LIN {X 0.040,Y -457.437,Z 279.553,A 0.000,B 0.000,C 90.000,E1 279.500} C_DIS
LIN {X 0.163,Y -463.352,Z 279.547,A 0.000,B 0.000,C 90.000,E1 278.454} C_DIS
LIN {X -0.027,Y -471.556,Z 279.539,A 0.000,B 0.000,C 90.000,E1 276.947} C_DIS
LIN {X 0.196,Y -476.547,Z 279.533,A 0.000,B 0.000,C 90.000,E1 275.910} C_DIS
LIN {X -0.146,Y -478.748,Z 279.530,A 0.000,B 0.000,C 90.000,E1 275.448} C_DIS
LIN {X -0.043,Y -480.665,Z 279.527,A 0.000,B 0.000,C 90.000,E1 274.935} C_DIS
LIN {X 0.113,Y -482.200,Z 279.525,A 0.000,B 0.000,C 90.000,E1 274.416} C_DIS
LIN {X -0.205,Y -483.358,Z 279.522,A 0.000,B 0.000,C 90.000,E1 273.955} C_DIS
LIN {X -0.065,Y -484.126,Z 279.519,A 0.000,B 0.000,C 90.000,E1 273.440} C_DIS
LIN {X 0.111,Y -484.567,Z 279.516,A 0.000,B 0.000,C 90.000,E1 272.922} C_DIS
LIN {X -0.218,Y -484.699,Z 279.514,A 0.000,B 0.000,C 90.000,E1 272.465} C_DIS
LIN {X 0.119,Y -484.413,Z 279.508,A 0.000,B 0.000,C 90.000,E1 271.432} C_DIS
LIN {X -0.203,Y -484.109,Z 279.505,A 0.000,B 0.000,C 90.000,E1 270.974} C_DIS
LIN {X -0.042,Y -483.584,Z 279.503,A 0.000,B 0.000,C 90.000,E1 270.458} C_DIS
LIN {X 0.119,Y -482.708,Z 279.500,A 0.000,B 0.000,C 90.000,E1 269.943} C_DIS
LIN {X -0.206,Y -481.433,Z 279.497,A 0.000,B 0.000,C 90.000,E1 269.484} C_DIS
LIN {X -0.056,Y -479.640,Z 279.494,A 0.000,B 0.000,C 90.000,E1 268.969} C_DIS
LIN {X 0.085,Y -477.139,Z 279.491,A 0.000,B 0.000,C 90.000,E1 268.453} C_DIS
LIN {X 0.223,Y -473.997,Z 279.489,A 0.000,B 0.000,C 90.000,E1 267.936} C_DIS
LIN {X -0.142,Y -469.925,Z 279.486,A 0.000,B 0.000,C 90.000,E1 267.478} C_DIS
LIN {X 0.134,Y -467.510,Z 279.484,A 0.000,B 0.000,C 90.000,E1 267.192} C_DIS
LIN {X -0.099,Y -461.974,Z 279.482,A 0.000,B 0.000,C 90.000,E1 266.731} C_DIS
LIN {X -0.164,Y -458.751,Z 279.480,A 0.000,B 0.000,C 90.000,E1 266.502} C_DIS
LIN {X 0.047,Y -455.605,Z 279.479,A 0.000,B 0.000,C 90.000,E1 266.274} C_DIS
LIN {X -0.198,Y -451.886,Z 279.478,A 0.000,B 0.000,C 90.000,E1 266.102} C_DIS
LIN {X -0.075,Y -448.465,Z 279.477,A 0.000,B 0.000,C 90.000,E1 265.927} C_DIS
LIN {X 0.016,Y -444.357,Z 279.476,A 0.000,B 0.000,C 90.000,E1 265.755} C_DIS
LIN {X -0.022,Y -440.666,Z 279.476,A 0.000,B 0.000,C 90.000,E1 265.641} C_DIS
LIN {X -0.059,Y -435.858,Z 279.475,A 0.000,B 0.000,C 90.000,E1 265.527} C_DIS
LIN {X 0.058,Y -425.990,Z 279.474,A 0.000,B 0.000,C 90.000,E1 265.355} C_DIS
LIN {X 0.041,Y -418.591,Z 279.474,A 0.000,B 0.000,C 90.000,E1 265.298} C_DIS
LIN {X -0.001,Y -180.904,Z 279.474,A 0.000,B 0.000,C 90.000,E1 265.298} C_DIS
LIN {X 0.035,Y -180.229,Z 279.464,A 0.000,B 0.000,C 90.000,E1 263.571} C_DIS
LIN {X -0.012,Y -179.042,Z 279.446,A 0.000,B 0.000,C 90.000,E1 260.208} C_DIS
LIN {X 0.051,Y -178.713,Z 279.441,A 0.000,B 0.000,C 90.000,E1 259.342} C_DIS
LIN {X -0.056,Y -175.761,Z 279.413,A 0.000,B 0.000,C 90.000,E1 254.283} C_DIS
LIN {X -0.006,Y -171.945,Z 279.384,A 0.000,B 0.000,C 90.000,E1 249.135} C_DIS
LIN {X -0.030,Y -171.330,Z 279.379,A 0.000,B 0.000,C 90.000,E1 248.284} C_DIS
LIN {X 0.022,Y -167.585,Z 279.355,A 0.000,B 0.000,C 90.000,E1 243.948} C_DIS
LIN {X -0.039,Y -166.222,Z 279.346,A 0.000,B 0.000,C 90.000,E1 242.231} C_DIS
LIN {X -0.050,Y -162.984,Z 279.326,A 0.000,B 0.000,C 90.000,E1 238.742} C_DIS
LIN {X -0.003,Y -160.899,Z 279.312,A 0.000,B 0.000,C 90.000,E1 236.087} C_DIS
LIN {X -0.025,Y -157.667,Z 279.292,A 0.000,B 0.000,C 90.000,E1 232.557} C_DIS
LIN {X -0.086,Y -155.705,Z 279.277,A 0.000,B 0.000,C 90.000,E1 229.908} C_DIS
LIN {X -0.032,Y -151.967,Z 279.252,A 0.000,B 0.000,C 90.000,E1 225.405} C_DIS
LIN {X -0.015,Y -150.210,Z 279.237,A 0.000,B 0.000,C 90.000,E1 222.690} C_DIS
LIN {X -0.090,Y -146.976,Z 279.212,A 0.000,B 0.000,C 90.000,E1 218.177} C_DIS
LIN {X 0.019,Y -145.562,Z 279.197,A 0.000,B 0.000,C 90.000,E1 215.391} C_DIS
LIN {X 0.018,Y -142.954,Z 279.171,A 0.000,B 0.000,C 90.000,E1 210.797} C_DIS
LIN {X -0.051,Y -141.580,Z 279.151,A 0.000,B 0.000,C 90.000,E1 207.129} C_DIS
LIN {X -0.003,Y -139.415,Z 279.115,A 0.000,B 0.000,C 90.000,E1 200.610} C_DIS
LIN {X 0.048,Y -139.140,Z 279.104,A 0.000,B 0.000,C 90.000,E1 198.725} C_DIS
LIN {X -0.061,Y -138.348,Z 279.057,A 0.000,B 0.000,C 90.000,E1 190.366} C_DIS
LIN {X 0.063,Y -139.492,Z 279.006,A 0.000,B 0.000,C 90.000,E1 180.974} C_DIS
LIN {X 0.004,Y -141.103,Z 278.975,A 0.000,B 0.000,C 90.000,E1 175.412} C_DIS
LIN {X -0.043,Y -142.482,Z 278.959,A 0.000,B 0.000,C 90.000,E1 172.648} C_DIS
LIN {X 0.047,Y -144.731,Z 278.933,A 0.000,B 0.000,C 90.000,E1 167.993} C_DIS
LIN {X -0.003,Y -147.335,Z 278.913,A 0.000,B 0.000,C 90.000,E1 164.338} C_DIS
LIN {X 0.062,Y -150.658,Z 278.888,A 0.000,B 0.000,C 90.000,E1 159.752} C_DIS
LIN {X -0.056,Y -154.136,Z 278.868,A 0.000,B 0.000,C 90.000,E1 156.177} C_DIS
LIN {X 0.006,Y -157.565,Z 278.848,A 0.000,B 0.000,C 90.000,E1 152.564} C_DIS
LIN {X 0.030,Y -161.808,Z 278.828,A 0.000,B 0.000,C 90.000,E1 148.997} C_DIS
LIN {X 0.050,Y -166.000,Z 278.808,A 0.000,B 0.000,C 90.000,E1 145.468} C_DIS
LIN {X 0.042,Y -170.999,Z 278.789,A 0.000,B 0.000,C 90.000,E1 141.984} C_DIS
LIN {X -0.042,Y -175.868,Z 278.770,A 0.000,B 0.000,C 90.000,E1 138.566} C_DIS
LIN {X -0.049,Y -181.473,Z 278.751,A 0.000,B 0.000,C 90.000,E1 135.162} C_DIS
LIN {X 0.088,Y -186.986,Z 278.732,A 0.000,B 0.000,C 90.000,E1 131.757} C_DIS
LIN {X 0.090,Y -190.102,Z 278.723,A 0.000,B 0.000,C 90.000,E1 130.092} C_DIS
LIN {X 0.110,Y -195.874,Z 278.705,A 0.000,B 0.000,C 90.000,E1 126.790} C_DIS
LIN {X -0.098,Y -200.705,Z 278.691,A 0.000,B 0.000,C 90.000,E1 124.405} C_DIS
LIN {X 0.009,Y -203.178,Z 278.683,A 0.000,B 0.000,C 90.000,E1 122.959} C_DIS
LIN {X -0.023,Y -305.671,Z 278.683,A 0.000,B 0.000,C 90.000,E1 122.959} C_DIS
LIN {X 0.050,Y -311.024,Z 278.682,A 0.000,B 0.000,C 90.000,E1 122.752} C_DIS
LIN {X 0.065,Y -314.178,Z 278.681,A 0.000,B 0.000,C 90.000,E1 122.498} C_DIS
LIN {X -0.074,Y -317.883,Z 278.678,A 0.000,B 0.000,C 90.000,E1 122.054} C_DIS
LIN {X -0.012,Y -319.669,Z 278.676,A 0.000,B 0.000,C 90.000,E1 121.720} C_DIS
LIN {X -0.034,Y -322.247,Z 278.673,A 0.000,B 0.000,C 90.000,E1 121.082} C_DIS
LIN {X -0.019,Y -333.580,Z 278.657,A 0.000,B 0.000,C 90.000,E1 118.231} C_DIS
LIN {X -0.161,Y -346.345,Z 278.641,A 0.000,B 0.000,C 90.000,E1 115.463} C_DIS
LIN {X -0.119,Y -358.992,Z 278.628,A 0.000,B 0.000,C 90.000,E1 113.025} C_DIS
LIN {X 0.117,Y -372.959,Z 278.615,A 0.000,B 0.000,C 90.000,E1 110.610} C_DIS
LIN {X -0.037,Y -388.346,Z 278.602,A 0.000,B 0.000,C 90.000,E1 108.308} C_DIS
LIN {X 0.072,Y -405.270,Z 278.589,A 0.000,B 0.000,C 90.000,E1 106.024} C_DIS
LIN {X -0.019,Y -423.855,Z 278.577,A 0.000,B 0.000,C 90.000,E1 103.828} C_DIS
LIN {X 0.042,Y -443.818,Z 278.565,A 0.000,B 0.000,C 90.000,E1 101.715} C_DIS
LIN {X -0.025,Y -464.375,Z 278.554,A 0.000,B 0.000,C 90.000,E1 99.792} C_DIS
LIN {X -0.069,Y -488.109,Z 278.543,A 0.000,B 0.000,C 90.000,E1 97.814} C_DIS
LIN {X 0.073,Y -501.323,Z 278.538,A 0.000,B 0.000,C 90.000,E1 96.777} C_DIS
LIN {X -0.176,Y -503.227,Z 278.537,A 0.000,B 0.000,C 90.000,E1 96.606} C_DIS
LIN {X 0.250,Y -504.994,Z 278.535,A 0.000,B 0.000,C 90.000,E1 96.315} C_DIS
LIN {X 0.120,Y -506.320,Z 278.534,A 0.000,B 0.000,C 90.000,E1 96.087} C_DIS
LIN {X -0.066,Y -507.964,Z 278.531,A 0.000,B 0.000,C 90.000,E1 95.625} C_DIS
LIN {X -0.247,Y -508.512,Z 278.529,A 0.000,B 0.000,C 90.000,E1 95.163} C_DIS
LIN {X 0.086,Y -508.054,Z 278.526,A 0.000,B 0.000,C 90.000,E1 94.645} C_DIS
LIN {X -0.125,Y -506.510,Z 278.523,A 0.000,B 0.000,C 90.000,E1 94.188} C_DIS
LIN {X -0.194,Y -505.243,Z 278.522,A 0.000,B 0.000,C 90.000,E1 93.955} C_DIS
LIN {X 0.093,Y -501.741,Z 278.519,A 0.000,B 0.000,C 90.000,E1 93.440} C_DIS
LIN {X 0.140,Y -493.907,Z 278.514,A 0.000,B 0.000,C 90.000,E1 92.465} C_DIS
LIN {X -0.053,Y -483.305,Z 278.507,A 0.000,B 0.000,C 90.000,E1 91.260} C_DIS
LIN {X -0.212,Y -464.590,Z 278.494,A 0.000,B 0.000,C 90.000,E1 89.026} C_DIS
LIN {X 0.122,Y -451.376,Z 278.484,A 0.000,B 0.000,C 90.000,E1 87.192} C_DIS
LIN {X 0.186,Y -430.844,Z 278.467,A 0.000,B 0.000,C 90.000,E1 84.033} C_DIS
LIN {X -0.180,Y -416.871,Z 278.454,A 0.000,B 0.000,C 90.000,E1 81.659} C_DIS
LIN {X 0.002,Y -404.089,Z 278.440,A 0.000,B 0.000,C 90.000,E1 79.162} C_DIS
LIN {X -0.157,Y -394.044,Z 278.429,A 0.000,B 0.000,C 90.000,E1 77.229} C_DIS
LIN {X -0.017,Y -382.646,Z 278.416,A 0.000,B 0.000,C 90.000,E1 74.936} C_DIS
LIN {X 0.035,Y -374.165,Z 278.407,A 0.000,B 0.000,C 90.000,E1 73.196} C_DIS
LIN {X -0.012,Y -362.792,Z 278.394,A 0.000,B 0.000,C 90.000,E1 70.859} C_DIS
LIN {X 0.068,Y -350.331,Z 278.379,A 0.000,B 0.000,C 90.000,E1 68.156} C_DIS
LIN {X 0.070,Y -336.135,Z 278.360,A 0.000,B 0.000,C 90.000,E1 64.793} C_DIS
LIN {X -0.024,Y -322.120,Z 278.339,A 0.000,B 0.000,C 90.000,E1 61.051} C_DIS
LIN {X 0.127,Y -314.316,Z 278.327,A 0.000,B 0.000,C 90.000,E1 58.791} C_DIS
LIN {X 0.061,Y -305.742,Z 278.312,A 0.000,B 0.000,C 90.000,E1 56.215} C_DIS
LIN {X -0.112,Y -297.454,Z 278.298,A 0.000,B 0.000,C 90.000,E1 53.623} C_DIS
LIN {X 0.045,Y -289.244,Z 278.283,A 0.000,B 0.000,C 90.000,E1 50.928} C_DIS
LIN {X -0.099,Y -283.046,Z 278.272,A 0.000,B 0.000,C 90.000,E1 48.933} C_DIS
LIN {X 0.000,Y -272.943,Z 278.253,A 0.000,B 0.000,C 90.000,E1 45.486} C_DIS
LIN {X 0.038,Y -265.369,Z 278.237,A 0.000,B 0.000,C 90.000,E1 42.690} C_DIS
LIN {X -0.178,Y -259.814,Z 278.225,A 0.000,B 0.000,C 90.000,E1 40.620} C_DIS
LIN {X -0.101,Y -254.173,Z 278.214,A 0.000,B 0.000,C 90.000,E1 38.463} C_DIS
LIN {X -0.091,Y -248.423,Z 278.202,A 0.000,B 0.000,C 90.000,E1 36.297} C_DIS
LIN {X 0.064,Y -242.506,Z 278.189,A 0.000,B 0.000,C 90.000,E1 34.072} C_DIS
LIN {X -0.015,Y -232.916,Z 278.169,A 0.000,B 0.000,C 90.000,E1 30.384} C_DIS
LIN {X -0.085,Y -225.892,Z 278.152,A 0.000,B 0.000,C 90.000,E1 27.385} C_DIS
LIN {X -0.125,Y -219.659,Z 278.135,A 0.000,B 0.000,C 90.000,E1 24.335} C_DIS
LIN {X -0.029,Y -212.898,Z 278.113,A 0.000,B 0.000,C 90.000,E1 20.429} C_DIS
LIN {X -0.041,Y -207.094,Z 278.092,A 0.000,B 0.000,C 90.000,E1 16.496} C_DIS
LIN {X 0.077,Y -202.346,Z 278.069,A 0.000,B 0.000,C 90.000,E1 12.479} C_DIS
LIN {X 0.079,Y -198.629,Z 278.047,A 0.000,B 0.000,C 90.000,E1 8.454} C_DIS
LIN {X -0.050,Y -195.024,Z 278.016,A 0.000,B 0.000,C 90.000,E1 2.808} C_DIS
LIN {X 0.076,Y -195.799,Z 277.920,A 0.000,B 0.000,C 90.000,E1 345.589} C_DIS
LIN {X -0.008,Y -199.281,Z 277.893,A 0.000,B 0.000,C 90.000,E1 340.732} C_DIS
LIN {X 0.093,Y -203.362,Z 277.871,A 0.000,B 0.000,C 90.000,E1 336.666} C_DIS
LIN {X 0.003,Y -208.478,Z 277.848,A 0.000,B 0.000,C 90.000,E1 332.692} C_DIS
LIN {X -0.007,Y -214.658,Z 277.826,A 0.000,B 0.000,C 90.000,E1 328.742} C_DIS
LIN {X 0.080,Y -220.531,Z 277.809,A 0.000,B 0.000,C 90.000,E1 325.595} C_DIS
LIN {X -0.106,Y -227.213,Z 277.792,A 0.000,B 0.000,C 90.000,E1 322.557} C_DIS
LIN {X 0.076,Y -235.809,Z 277.773,A 0.000,B 0.000,C 90.000,E1 319.094} C_DIS
LIN {X 0.137,Y -245.410,Z 277.754,A 0.000,B 0.000,C 90.000,E1 315.729} C_DIS
LIN {X 0.135,Y -256.023,Z 277.736,A 0.000,B 0.000,C 90.000,E1 312.447} C_DIS
LIN {X -0.070,Y -267.676,Z 277.718,A 0.000,B 0.000,C 90.000,E1 309.277} C_DIS
LIN {X 0.151,Y -280.621,Z 277.701,A 0.000,B 0.000,C 90.000,E1 306.091} C_DIS
LIN {X 0.116,Y -293.578,Z 277.686,A 0.000,B 0.000,C 90.000,E1 303.372} C_DIS
LIN {X -0.041,Y -309.906,Z 277.669,A 0.000,B 0.000,C 90.000,E1 300.413} C_DIS
LIN {X 0.048,Y -329.857,Z 277.651,A 0.000,B 0.000,C 90.000,E1 297.180} C_DIS
LIN {X -0.144,Y -342.555,Z 277.641,A 0.000,B 0.000,C 90.000,E1 295.335} C_DIS
LIN {X 0.074,Y -355.273,Z 277.630,A 0.000,B 0.000,C 90.000,E1 293.462} C_DIS
LIN {X 0.079,Y -368.073,Z 277.620,A 0.000,B 0.000,C 90.000,E1 291.663} C_DIS
LIN {X 0.078,Y -385.539,Z 277.607,A 0.000,B 0.000,C 90.000,E1 289.322} C_DIS
LIN {X 0.060,Y -401.077,Z 277.596,A 0.000,B 0.000,C 90.000,E1 287.330} C_DIS
LIN {X 0.024,Y -414.297,Z 277.587,A 0.000,B 0.000,C 90.000,E1 285.662} C_DIS
LIN {X -0.034,Y -425.272,Z 277.579,A 0.000,B 0.000,C 90.000,E1 284.300} C_DIS
LIN {X 0.039,Y -431.512,Z 277.575,A 0.000,B 0.000,C 90.000,E1 283.480} C_DIS
LIN {X 0.038,Y -439.105,Z 277.569,A 0.000,B 0.000,C 90.000,E1 282.411} C_DIS
LIN {X 0.163,Y -447.753,Z 277.562,A 0.000,B 0.000,C 90.000,E1 281.074} C_DIS
LIN {X -0.014,Y -455.691,Z 277.554,A 0.000,B 0.000,C 90.000,E1 279.792} C_DIS
LIN {X 0.089,Y -461.705,Z 277.549,A 0.000,B 0.000,C 90.000,E1 278.746} C_DIS
LIN {X 0.035,Y -468.676,Z 277.542,A 0.000,B 0.000,C 90.000,E1 277.473} C_DIS
LIN {X -0.186,Y -473.921,Z 277.536,A 0.000,B 0.000,C 90.000,E1 276.486} C_DIS
LIN {X 0.017,Y -478.571,Z 277.530,A 0.000,B 0.000,C 90.000,E1 275.454} C_DIS
LIN {X 0.166,Y -480.481,Z 277.528,A 0.000,B 0.000,C 90.000,E1 274.935} C_DIS
LIN {X -0.160,Y -482.031,Z 277.525,A 0.000,B 0.000,C 90.000,E1 274.473} C_DIS
LIN {X 0.002,Y -483.221,Z 277.522,A 0.000,B 0.000,C 90.000,E1 273.955} C_DIS
LIN {X 0.141,Y -483.997,Z 277.519,A 0.000,B 0.000,C 90.000,E1 273.440} C_DIS
LIN {X -0.167,Y -484.471,Z 277.516,A 0.000,B 0.000,C 90.000,E1 272.980} C_DIS
LIN {X -0.013,Y -484.651,Z 277.514,A 0.000,B 0.000,C 90.000,E1 272.465} C_DIS
LIN {X 0.148,Y -484.631,Z 277.511,A 0.000,B 0.000,C 90.000,E1 271.949} C_DIS
LIN {X 0.001,Y -484.162,Z 277.505,A 0.000,B 0.000,C 90.000,E1 270.974} C_DIS
LIN {X 0.163,Y -483.651,Z 277.503,A 0.000,B 0.000,C 90.000,E1 270.458} C_DIS
LIN {X -0.160,Y -482.807,Z 277.500,A 0.000,B 0.000,C 90.000,E1 270.000} C_DIS
LIN {X -0.002,Y -481.535,Z 277.497,A 0.000,B 0.000,C 90.000,E1 269.484} C_DIS
LIN {X 0.148,Y -479.754,Z 277.494,A 0.000,B 0.000,C 90.000,E1 268.969} C_DIS
LIN {X -0.188,Y -477.339,Z 277.492,A 0.000,B 0.000,C 90.000,E1 268.511} C_DIS
LIN {X -0.048,Y -474.199,Z 277.489,A 0.000,B 0.000,C 90.000,E1 267.993} C_DIS
LIN {X 0.061,Y -470.202,Z 277.486,A 0.000,B 0.000,C 90.000,E1 267.478} C_DIS
LIN {X 0.143,Y -465.186,Z 277.483,A 0.000,B 0.000,C 90.000,E1 266.963} C_DIS
LIN {X 0.067,Y -462.356,Z 277.482,A 0.000,B 0.000,C 90.000,E1 266.731} C_DIS
LIN {X -0.032,Y -459.122,Z 277.481,A 0.000,B 0.000,C 90.000,E1 266.502} C_DIS
LIN {X 0.161,Y -455.979,Z 277.479,A 0.000,B 0.000,C 90.000,E1 266.274} C_DIS
LIN {X -0.003,Y -449.020,Z 277.477,A 0.000,B 0.000,C 90.000,E1 265.927} C_DIS
LIN {X 0.061,Y -444.993,Z 277.476,A 0.000,B 0.000,C 90.000,E1 265.755} C_DIS
LIN {X -0.081,Y -436.493,Z 277.475,A 0.000,B 0.000,C 90.000,E1 265.527} C_DIS
LIN {X 0.150,Y -432.276,Z 277.475,A 0.000,B 0.000,C 90.000,E1 265.412} C_DIS
LIN {X -0.049,Y -426.466,Z 277.474,A 0.000,B 0.000,C 90.000,E1 265.355} C_DIS
LIN {X -0.056,Y -419.057,Z 277.474,A 0.000,B 0.000,C 90.000,E1 265.298} C_DIS
LIN {X -0.104,Y -416.418,Z 277.474,A 0.000,B 0.000,C 90.000,E1 265.298} C_DIS
LIN {X -0.066,Y -180.902,Z 277.474,A 0.000,B 0.000,C 90.000,E1 265.298} C_DIS
LIN {X -0.018,Y -180.222,Z 277.464,A 0.000,B 0.000,C 90.000,E1 263.571} C_DIS
LIN {X -0.065,Y -179.037,Z 277.445,A 0.000,B 0.000,C 90.000,E1 260.208} C_DIS
LIN {X -0.002,Y -178.701,Z 277.441,A 0.000,B 0.000,C 90.000,E1 259.342} C_DIS
LIN {X -0.061,Y -175.751,Z 277.412,A 0.000,B 0.000,C 90.000,E1 254.267} C_DIS
LIN {X -0.058,Y -171.934,Z 277.384,A 0.000,B 0.000,C 90.000,E1 249.135} C_DIS
LIN {X -0.082,Y -171.314,Z 277.379,A 0.000,B 0.000,C 90.000,E1 248.284} C_DIS
LIN {X -0.028,Y -167.573,Z 277.355,A 0.000,B 0.000,C 90.000,E1 243.948} C_DIS
LIN {X -0.089,Y -166.203,Z 277.346,A 0.000,B 0.000,C 90.000,E1 242.231} C_DIS
LIN {X -0.100,Y -162.969,Z 277.326,A 0.000,B 0.000,C 90.000,E1 238.742} C_DIS
LIN {X -0.052,Y -160.881,Z 277.311,A 0.000,B 0.000,C 90.000,E1 236.087} C_DIS
LIN {X -0.073,Y -157.652,Z 277.292,A 0.000,B 0.000,C 90.000,E1 232.557} C_DIS
LIN {X 0.085,Y -155.689,Z 277.277,A 0.000,B 0.000,C 90.000,E1 229.828} C_DIS
LIN {X -0.079,Y -151.955,Z 277.252,A 0.000,B 0.000,C 90.000,E1 225.405} C_DIS
LIN {X -0.062,Y -150.195,Z 277.237,A 0.000,B 0.000,C 90.000,E1 222.690} C_DIS
LIN {X 0.069,Y -146.965,Z 277.212,A 0.000,B 0.000,C 90.000,E1 218.096} C_DIS
LIN {X -0.028,Y -145.552,Z 277.197,A 0.000,B 0.000,C 90.000,E1 215.391} C_DIS
LIN {X -0.028,Y -142.945,Z 277.171,A 0.000,B 0.000,C 90.000,E1 210.797} C_DIS
LIN {X 0.029,Y -141.571,Z 277.150,A 0.000,B 0.000,C 90.000,E1 207.078} C_DIS
LIN {X -0.049,Y -139.412,Z 277.114,A 0.000,B 0.000,C 90.000,E1 200.610} C_DIS
LIN {X 0.003,Y -139.135,Z 277.104,A 0.000,B 0.000,C 90.000,E1 198.725} C_DIS
LIN {X 0.030,Y -138.349,Z 277.057,A 0.000,B 0.000,C 90.000,E1 190.310} C_DIS
LIN {X 0.018,Y -139.494,Z 277.005,A 0.000,B 0.000,C 90.000,E1 180.974} C_DIS
LIN {X -0.042,Y -141.110,Z 276.974,A 0.000,B 0.000,C 90.000,E1 175.412} C_DIS
LIN {X 0.052,Y -142.490,Z 276.959,A 0.000,B 0.000,C 90.000,E1 172.591} C_DIS
LIN {X 0.000,Y -144.742,Z 276.933,A 0.000,B 0.000,C 90.000,E1 167.993} C_DIS
LIN {X -0.050,Y -147.349,Z 276.913,A 0.000,B 0.000,C 90.000,E1 164.338} C_DIS
LIN {X 0.014,Y -150.674,Z 276.888,A 0.000,B 0.000,C 90.000,E1 159.752} C_DIS
LIN {X 0.035,Y -154.154,Z 276.867,A 0.000,B 0.000,C 90.000,E1 156.125} C_DIS
LIN {X 0.029,Y -157.584,Z 276.848,A 0.000,B 0.000,C 90.000,E1 152.538} C_DIS
LIN {X -0.020,Y -161.832,Z 276.828,A 0.000,B 0.000,C 90.000,E1 148.997} C_DIS
LIN {X -0.001,Y -166.023,Z 276.808,A 0.000,B 0.000,C 90.000,E1 145.468} C_DIS
LIN {X -0.009,Y -171.024,Z 276.789,A 0.000,B 0.000,C 90.000,E1 141.984} C_DIS
LIN {X 0.022,Y -175.894,Z 276.770,A 0.000,B 0.000,C 90.000,E1 138.528} C_DIS
LIN {X 0.026,Y -181.499,Z 276.751,A 0.000,B 0.000,C 90.000,E1 135.121} C_DIS
LIN {X 0.033,Y -187.016,Z 276.732,A 0.000,B 0.000,C 90.000,E1 131.757} C_DIS
LIN {X 0.035,Y -190.134,Z 276.723,A 0.000,B 0.000,C 90.000,E1 130.092} C_DIS
LIN {X 0.053,Y -195.905,Z 276.704,A 0.000,B 0.000,C 90.000,E1 126.790} C_DIS
LIN {X 0.010,Y -200.736,Z 276.691,A 0.000,B 0.000,C 90.000,E1 124.358} C_DIS
LIN {X 0.023,Y -203.258,Z 276.683,A 0.000,B 0.000,C 90.000,E1 122.911} C_DIS
LIN {X 0.166,Y -305.477,Z 276.683,A 0.000,B 0.000,C 90.000,E1 122.880} C_DIS
LIN {X 0.096,Y -306.527,Z 276.683,A 0.000,B 0.000,C 90.000,E1 122.880} C_DIS
LIN {X -0.037,Y -310.653,Z 276.682,A 0.000,B 0.000,C 90.000,E1 122.752} C_DIS
LIN {X -0.175,Y -313.783,Z 276.681,A 0.000,B 0.000,C 90.000,E1 122.546} C_DIS
LIN {X -0.051,Y -317.498,Z 276.678,A 0.000,B 0.000,C 90.000,E1 122.084} C_DIS
LIN {X 0.045,Y -319.375,Z 276.676,A 0.000,B 0.000,C 90.000,E1 121.750} C_DIS
LIN {X -0.131,Y -320.846,Z 276.675,A 0.000,B 0.000,C 90.000,E1 121.465} C_DIS
LIN {X -0.050,Y -333.366,Z 276.657,A 0.000,B 0.000,C 90.000,E1 118.281} C_DIS
LIN {X 0.106,Y -346.106,Z 276.642,A 0.000,B 0.000,C 90.000,E1 115.463} C_DIS
LIN {X -0.179,Y -358.730,Z 276.628,A 0.000,B 0.000,C 90.000,E1 113.078} C_DIS
LIN {X 0.042,Y -372.672,Z 276.615,A 0.000,B 0.000,C 90.000,E1 110.663} C_DIS
LIN {X -0.128,Y -388.033,Z 276.602,A 0.000,B 0.000,C 90.000,E1 108.362} C_DIS
LIN {X -0.035,Y -404.928,Z 276.589,A 0.000,B 0.000,C 90.000,E1 106.079} C_DIS
LIN {X -0.145,Y -423.483,Z 276.577,A 0.000,B 0.000,C 90.000,E1 103.883} C_DIS
LIN {X -0.117,Y -443.431,Z 276.565,A 0.000,B 0.000,C 90.000,E1 101.771} C_DIS
LIN {X -0.219,Y -463.979,Z 276.555,A 0.000,B 0.000,C 90.000,E1 99.849} C_DIS
LIN {X 0.181,Y -487.703,Z 276.544,A 0.000,B 0.000,C 90.000,E1 97.814} C_DIS
LIN {X -0.181,Y -501.020,Z 276.538,A 0.000,B 0.000,C 90.000,E1 96.834} C_DIS
LIN {X 0.065,Y -503.054,Z 276.537,A 0.000,B 0.000,C 90.000,E1 96.606} C_DIS
LIN {X 0.034,Y -504.896,Z 276.535,A 0.000,B 0.000,C 90.000,E1 96.372} C_DIS
LIN {X -0.055,Y -506.285,Z 276.534,A 0.000,B 0.000,C 90.000,E1 96.144} C_DIS
LIN {X -0.242,Y -508.074,Z 276.531,A 0.000,B 0.000,C 90.000,E1 95.682} C_DIS
LIN {X 0.083,Y -508.746,Z 276.529,A 0.000,B 0.000,C 90.000,E1 95.163} C_DIS
LIN {X -0.092,Y -508.408,Z 276.526,A 0.000,B 0.000,C 90.000,E1 94.702} C_DIS
LIN {X 0.205,Y -507.003,Z 276.523,A 0.000,B 0.000,C 90.000,E1 94.188} C_DIS
LIN {X 0.137,Y -505.824,Z 276.522,A 0.000,B 0.000,C 90.000,E1 93.955} C_DIS
LIN {X -0.077,Y -502.412,Z 276.519,A 0.000,B 0.000,C 90.000,E1 93.498} C_DIS
LIN {X -0.021,Y -494.605,Z 276.514,A 0.000,B 0.000,C 90.000,E1 92.522} C_DIS
LIN {X -0.056,Y -486.151,Z 276.509,A 0.000,B 0.000,C 90.000,E1 91.547} C_DIS
LIN {X 0.127,Y -465.225,Z 276.495,A 0.000,B 0.000,C 90.000,E1 89.026} C_DIS
LIN {X -0.224,Y -450.154,Z 276.483,A 0.000,B 0.000,C 90.000,E1 87.020} C_DIS
LIN {X -0.144,Y -429.761,Z 276.466,A 0.000,B 0.000,C 90.000,E1 83.856} C_DIS
LIN {X -0.159,Y -415.912,Z 276.452,A 0.000,B 0.000,C 90.000,E1 81.432} C_DIS
LIN {X 0.059,Y -403.177,Z 276.439,A 0.000,B 0.000,C 90.000,E1 78.926} C_DIS
LIN {X -0.049,Y -391.708,Z 276.426,A 0.000,B 0.000,C 90.000,E1 76.700} C_DIS
LIN {X 0.150,Y -378.968,Z 276.412,A 0.000,B 0.000,C 90.000,E1 74.102} C_DIS
LIN {X 0.117,Y -369.022,Z 276.401,A 0.000,B 0.000,C 90.000,E1 72.072} C_DIS
LIN {X 0.168,Y -357.769,Z 276.387,A 0.000,B 0.000,C 90.000,E1 69.699} C_DIS
LIN {X -0.035,Y -343.020,Z 276.369,A 0.000,B 0.000,C 90.000,E1 66.410} C_DIS
LIN {X 0.012,Y -329.504,Z 276.350,A 0.000,B 0.000,C 90.000,E1 62.999} C_DIS
LIN {X -0.165,Y -318.241,Z 276.332,A 0.000,B 0.000,C 90.000,E1 59.871} C_DIS
LIN {X -0.083,Y -308.414,Z 276.316,A 0.000,B 0.000,C 90.000,E1 56.962} C_DIS
LIN {X 0.061,Y -300.058,Z 276.302,A 0.000,B 0.000,C 90.000,E1 54.322} C_DIS
LIN {X -0.080,Y -291.814,Z 276.287,A 0.000,B 0.000,C 90.000,E1 51.698} C_DIS
LIN {X 0.006,Y -285.627,Z 276.276,A 0.000,B 0.000,C 90.000,E1 49.666} C_DIS
LIN {X 0.002,Y -277.354,Z 276.261,A 0.000,B 0.000,C 90.000,E1 46.944} C_DIS
LIN {X 0.101,Y -267.697,Z 276.242,A 0.000,B 0.000,C 90.000,E1 43.461} C_DIS
LIN {X -0.077,Y -262.136,Z 276.230,A 0.000,B 0.000,C 90.000,E1 41.391} C_DIS
LIN {X -0.153,Y -256.479,Z 276.218,A 0.000,B 0.000,C 90.000,E1 39.277} C_DIS
LIN {X 0.055,Y -250.786,Z 276.206,A 0.000,B 0.000,C 90.000,E1 37.076} C_DIS
LIN {X 0.050,Y -244.966,Z 276.194,A 0.000,B 0.000,C 90.000,E1 34.898} C_DIS
LIN {X 0.050,Y -235.268,Z 276.173,A 0.000,B 0.000,C 90.000,E1 31.209} C_DIS
LIN {X -0.048,Y -228.056,Z 276.157,A 0.000,B 0.000,C 90.000,E1 28.231} C_DIS
LIN {X 0.062,Y -221.574,Z 276.140,A 0.000,B 0.000,C 90.000,E1 25.155} C_DIS
LIN {X 0.095,Y -214.603,Z 276.118,A 0.000,B 0.000,C 90.000,E1 21.280} C_DIS
LIN {X -0.068,Y -208.573,Z 276.097,A 0.000,B 0.000,C 90.000,E1 17.402} C_DIS
LIN {X 0.002,Y -203.585,Z 276.075,A 0.000,B 0.000,C 90.000,E1 13.411} C_DIS
LIN {X 0.072,Y -199.616,Z 276.052,A 0.000,B 0.000,C 90.000,E1 9.378} C_DIS
LIN {X 0.031,Y -196.174,Z 276.025,A 0.000,B 0.000,C 90.000,E1 4.531} C_DIS
LIN {X 0.055,Y -193.687,Z 275.988,A 0.000,B 0.000,C 90.000,E1 357.879} C_DIS
LIN {X 0.074,Y -195.175,Z 275.929,A 0.000,B 0.000,C 90.000,E1 347.229} C_DIS
LIN {X -0.006,Y -198.134,Z 275.902,A 0.000,B 0.000,C 90.000,E1 342.362} C_DIS
LIN {X 0.102,Y -201.807,Z 275.880,A 0.000,B 0.000,C 90.000,E1 338.284} C_DIS
LIN {X 0.066,Y -206.458,Z 275.857,A 0.000,B 0.000,C 90.000,E1 334.280} C_DIS
LIN {X -0.021,Y -212.223,Z 275.835,A 0.000,B 0.000,C 90.000,E1 330.333} C_DIS
LIN {X 0.069,Y -217.700,Z 275.818,A 0.000,B 0.000,C 90.000,E1 327.168} C_DIS
LIN {X 0.052,Y -223.962,Z 275.800,A 0.000,B 0.000,C 90.000,E1 324.069} C_DIS
LIN {X 0.046,Y -231.155,Z 275.783,A 0.000,B 0.000,C 90.000,E1 321.009} C_DIS
LIN {X -0.004,Y -240.155,Z 275.765,A 0.000,B 0.000,C 90.000,E1 317.634} C_DIS
LIN {X 0.003,Y -250.210,Z 275.746,A 0.000,B 0.000,C 90.000,E1 314.312} C_DIS
LIN {X -0.032,Y -261.268,Z 275.728,A 0.000,B 0.000,C 90.000,E1 311.067} C_DIS
LIN {X -0.055,Y -273.468,Z 275.710,A 0.000,B 0.000,C 90.000,E1 307.890} C_DIS
LIN {X 0.045,Y -285.503,Z 275.695,A 0.000,B 0.000,C 90.000,E1 305.105} C_DIS
LIN {X -0.033,Y -299.038,Z 275.680,A 0.000,B 0.000,C 90.000,E1 302.418} C_DIS
LIN {X -0.035,Y -315.883,Z 275.664,A 0.000,B 0.000,C 90.000,E1 299.461} C_DIS
LIN {X -0.071,Y -336.353,Z 275.646,A 0.000,B 0.000,C 90.000,E1 296.283} C_DIS
LIN {X 0.169,Y -349.044,Z 275.636,A 0.000,B 0.000,C 90.000,E1 294.387} C_DIS
LIN {X 0.053,Y -361.782,Z 275.626,A 0.000,B 0.000,C 90.000,E1 292.589} C_DIS
LIN {X -0.101,Y -378.958,Z 275.612,A 0.000,B 0.000,C 90.000,E1 290.248} C_DIS
LIN {X 0.078,Y -392.195,Z 275.603,A 0.000,B 0.000,C 90.000,E1 288.489} C_DIS
LIN {X 0.007,Y -405.467,Z 275.593,A 0.000,B 0.000,C 90.000,E1 286.804} C_DIS
LIN {X -0.114,Y -420.807,Z 275.583,A 0.000,B 0.000,C 90.000,E1 284.883} C_DIS
LIN {X 0.070,Y -429.351,Z 275.577,A 0.000,B 0.000,C 90.000,E1 283.772} C_DIS
LIN {X -0.239,Y -435.258,Z 275.572,A 0.000,B 0.000,C 90.000,E1 283.008} C_DIS
LIN {X 0.136,Y -442.500,Z 275.566,A 0.000,B 0.000,C 90.000,E1 281.895} C_DIS
LIN {X 0.169,Y -449.217,Z 275.560,A 0.000,B 0.000,C 90.000,E1 280.838} C_DIS
LIN {X -0.178,Y -458.553,Z 275.552,A 0.000,B 0.000,C 90.000,E1 279.321} C_DIS
LIN {X 0.174,Y -465.737,Z 275.545,A 0.000,B 0.000,C 90.000,E1 277.992} C_DIS
LIN {X 0.181,Y -472.480,Z 275.537,A 0.000,B 0.000,C 90.000,E1 276.720} C_DIS
LIN {X -0.055,Y -477.305,Z 275.532,A 0.000,B 0.000,C 90.000,E1 275.739} C_DIS
LIN {X -0.103,Y -480.308,Z 275.528,A 0.000,B 0.000,C 90.000,E1 274.992} C_DIS
LIN {X 0.049,Y -481.904,Z 275.525,A 0.000,B 0.000,C 90.000,E1 274.473} C_DIS
LIN {X 0.210,Y -483.117,Z 275.522,A 0.000,B 0.000,C 90.000,E1 273.955} C_DIS
LIN {X -0.134,Y -483.951,Z 275.519,A 0.000,B 0.000,C 90.000,E1 273.498} C_DIS
LIN {X 0.041,Y -484.449,Z 275.517,A 0.000,B 0.000,C 90.000,E1 272.980} C_DIS
LIN {X 0.195,Y -484.646,Z 275.514,A 0.000,B 0.000,C 90.000,E1 272.465} C_DIS
LIN {X 0.048,Y -484.483,Z 275.508,A 0.000,B 0.000,C 90.000,E1 271.489} C_DIS
LIN {X 0.209,Y -484.243,Z 275.506,A 0.000,B 0.000,C 90.000,E1 270.974} C_DIS
LIN {X -0.114,Y -483.747,Z 275.503,A 0.000,B 0.000,C 90.000,E1 270.516} C_DIS
LIN {X 0.048,Y -482.939,Z 275.500,A 0.000,B 0.000,C 90.000,E1 270.000} C_DIS
LIN {X 0.205,Y -481.671,Z 275.497,A 0.000,B 0.000,C 90.000,E1 269.484} C_DIS
LIN {X -0.123,Y -479.933,Z 275.495,A 0.000,B 0.000,C 90.000,E1 269.026} C_DIS
LIN {X 0.020,Y -477.542,Z 275.492,A 0.000,B 0.000,C 90.000,E1 268.511} C_DIS
LIN {X 0.159,Y -474.440,Z 275.489,A 0.000,B 0.000,C 90.000,E1 267.993} C_DIS
LIN {X -0.203,Y -470.523,Z 275.486,A 0.000,B 0.000,C 90.000,E1 267.535} C_DIS
LIN {X -0.116,Y -465.534,Z 275.483,A 0.000,B 0.000,C 90.000,E1 267.020} C_DIS
LIN {X -0.194,Y -462.754,Z 275.482,A 0.000,B 0.000,C 90.000,E1 266.788} C_DIS
LIN {X 0.164,Y -459.614,Z 275.481,A 0.000,B 0.000,C 90.000,E1 266.502} C_DIS
LIN {X 0.016,Y -452.967,Z 275.478,A 0.000,B 0.000,C 90.000,E1 266.102} C_DIS
LIN {X 0.006,Y -445.200,Z 275.476,A 0.000,B 0.000,C 90.000,E1 265.755} C_DIS
LIN {X -0.093,Y -441.398,Z 275.476,A 0.000,B 0.000,C 90.000,E1 265.641} C_DIS
LIN {X -0.191,Y -436.575,Z 275.475,A 0.000,B 0.000,C 90.000,E1 265.527} C_DIS
LIN {X 0.049,Y -432.520,Z 275.475,A 0.000,B 0.000,C 90.000,E1 265.412} C_DIS
LIN {X -0.143,Y -426.900,Z 275.474,A 0.000,B 0.000,C 90.000,E1 265.355} C_DIS
LIN {X -0.152,Y -419.460,Z 275.474,A 0.000,B 0.000,C 90.000,E1 265.298} C_DIS
LIN {X -0.199,Y -414.845,Z 275.474,A 0.000,B 0.000,C 90.000,E1 265.298} C_DIS
LIN {X 0.072,Y -180.902,Z 275.474,A 0.000,B 0.000,C 90.000,E1 265.241} C_DIS
LIN {X -0.063,Y -180.215,Z 275.464,A 0.000,B 0.000,C 90.000,E1 263.571} C_DIS
LIN {X 0.067,Y -179.034,Z 275.445,A 0.000,B 0.000,C 90.000,E1 260.151} C_DIS
LIN {X -0.047,Y -178.693,Z 275.441,A 0.000,B 0.000,C 90.000,E1 259.342} C_DIS
LIN {X 0.064,Y -175.741,Z 275.412,A 0.000,B 0.000,C 90.000,E1 254.212} C_DIS
LIN {X 0.059,Y -171.925,Z 275.384,A 0.000,B 0.000,C 90.000,E1 249.082} C_DIS
LIN {X 0.034,Y -171.300,Z 275.379,A 0.000,B 0.000,C 90.000,E1 248.230} C_DIS
LIN {X 0.079,Y -167.562,Z 275.355,A 0.000,B 0.000,C 90.000,E1 243.896} C_DIS
LIN {X 0.092,Y -166.188,Z 275.345,A 0.000,B 0.000,C 90.000,E1 242.153} C_DIS
LIN {X 0.081,Y -162.957,Z 275.326,A 0.000,B 0.000,C 90.000,E1 238.663} C_DIS
LIN {X -0.095,Y -160.866,Z 275.311,A 0.000,B 0.000,C 90.000,E1 236.087} C_DIS
LIN {X 0.010,Y -157.640,Z 275.292,A 0.000,B 0.000,C 90.000,E1 232.512} C_DIS
LIN {X 0.043,Y -155.677,Z 275.277,A 0.000,B 0.000,C 90.000,E1 229.828} C_DIS
LIN {X -0.012,Y -151.943,Z 275.252,A 0.000,B 0.000,C 90.000,E1 225.364} C_DIS
LIN {X -0.103,Y -150.183,Z 275.237,A 0.000,B 0.000,C 90.000,E1 222.690} C_DIS
LIN {X 0.029,Y -146.956,Z 275.212,A 0.000,B 0.000,C 90.000,E1 218.096} C_DIS
LIN {X -0.068,Y -145.544,Z 275.196,A 0.000,B 0.000,C 90.000,E1 215.391} C_DIS
LIN {X -0.067,Y -142.939,Z 275.171,A 0.000,B 0.000,C 90.000,E1 210.797} C_DIS
LIN {X -0.010,Y -141.563,Z 275.150,A 0.000,B 0.000,C 90.000,E1 207.078} C_DIS
LIN {X 0.043,Y -139.409,Z 275.114,A 0.000,B 0.000,C 90.000,E1 200.556} C_DIS
LIN {X -0.035,Y -139.131,Z 275.104,A 0.000,B 0.000,C 90.000,E1 198.725} C_DIS
LIN {X -0.008,Y -138.350,Z 275.057,A 0.000,B 0.000,C 90.000,E1 190.310} C_DIS
LIN {X -0.021,Y -139.497,Z 275.005,A 0.000,B 0.000,C 90.000,E1 180.974} C_DIS
LIN {X 0.060,Y -141.118,Z 274.974,A 0.000,B 0.000,C 90.000,E1 175.355} C_DIS
LIN {X 0.014,Y -142.497,Z 274.959,A 0.000,B 0.000,C 90.000,E1 172.591} C_DIS
LIN {X -0.040,Y -144.752,Z 274.933,A 0.000,B 0.000,C 90.000,E1 167.993} C_DIS
LIN {X 0.052,Y -147.361,Z 274.913,A 0.000,B 0.000,C 90.000,E1 164.283} C_DIS
LIN {X -0.026,Y -150.688,Z 274.887,A 0.000,B 0.000,C 90.000,E1 159.752} C_DIS
LIN {X 0.057,Y -154.168,Z 274.867,A 0.000,B 0.000,C 90.000,E1 156.102} C_DIS
LIN {X -0.013,Y -157.600,Z 274.847,A 0.000,B 0.000,C 90.000,E1 152.538} C_DIS
LIN {X -0.063,Y -161.852,Z 274.828,A 0.000,B 0.000,C 90.000,E1 148.997} C_DIS
LIN {X -0.045,Y -166.043,Z 274.808,A 0.000,B 0.000,C 90.000,E1 145.468} C_DIS
LIN {X -0.053,Y -171.045,Z 274.789,A 0.000,B 0.000,C 90.000,E1 141.984} C_DIS
LIN {X -0.024,Y -175.917,Z 274.770,A 0.000,B 0.000,C 90.000,E1 138.528} C_DIS
LIN {X -0.031,Y -180.155,Z 274.755,A 0.000,B 0.000,C 90.000,E1 135.972} C_DIS
LIN {X -0.062,Y -185.573,Z 274.737,A 0.000,B 0.000,C 90.000,E1 132.609} C_DIS
LIN {X -0.012,Y -190.161,Z 274.723,A 0.000,B 0.000,C 90.000,E1 130.092} C_DIS
LIN {X 0.033,Y -197.490,Z 274.700,A 0.000,B 0.000,C 90.000,E1 125.964} C_DIS
LIN {X 0.075,Y -200.761,Z 274.691,A 0.000,B 0.000,C 90.000,E1 124.326} C_DIS
LIN {X -0.038,Y -203.345,Z 274.683,A 0.000,B 0.000,C 90.000,E1 122.880} C_DIS
LIN {X -0.091,Y -305.482,Z 274.683,A 0.000,B 0.000,C 90.000,E1 122.880} C_DIS
LIN {X -0.112,Y -310.139,Z 274.682,A 0.000,B 0.000,C 90.000,E1 122.752} C_DIS
LIN {X -0.066,Y -313.140,Z 274.681,A 0.000,B 0.000,C 90.000,E1 122.546} C_DIS
LIN {X 0.021,Y -316.867,Z 274.679,A 0.000,B 0.000,C 90.000,E1 122.133} C_DIS
LIN {X -0.028,Y -318.799,Z 274.677,A 0.000,B 0.000,C 90.000,E1 121.848} C_DIS
LIN {X 0.026,Y -320.323,Z 274.675,A 0.000,B 0.000,C 90.000,E1 121.544} C_DIS
LIN {X -0.168,Y -327.727,Z 274.665,A 0.000,B 0.000,C 90.000,E1 119.667} C_DIS
LIN {X -0.022,Y -339.764,Z 274.649,A 0.000,B 0.000,C 90.000,E1 116.821} C_DIS
LIN {X 0.154,Y -351.713,Z 274.635,A 0.000,B 0.000,C 90.000,E1 114.335} C_DIS
LIN {X -0.126,Y -364.929,Z 274.622,A 0.000,B 0.000,C 90.000,E1 111.972} C_DIS
LIN {X 0.129,Y -379.508,Z 274.609,A 0.000,B 0.000,C 90.000,E1 109.577} C_DIS
LIN {X 0.140,Y -395.557,Z 274.596,A 0.000,B 0.000,C 90.000,E1 107.275} C_DIS
LIN {X -0.081,Y -413.196,Z 274.584,A 0.000,B 0.000,C 90.000,E1 105.064} C_DIS
LIN {X -0.061,Y -432.517,Z 274.572,A 0.000,B 0.000,C 90.000,E1 102.883} C_DIS
LIN {X 0.071,Y -452.766,Z 274.560,A 0.000,B 0.000,C 90.000,E1 100.838} C_DIS
LIN {X 0.131,Y -473.552,Z 274.550,A 0.000,B 0.000,C 90.000,E1 98.973} C_DIS
LIN {X 0.088,Y -497.509,Z 274.539,A 0.000,B 0.000,C 90.000,E1 97.068} C_DIS
LIN {X -0.108,Y -500.188,Z 274.538,A 0.000,B 0.000,C 90.000,E1 96.891} C_DIS
LIN {X 0.133,Y -502.497,Z 274.537,A 0.000,B 0.000,C 90.000,E1 96.663} C_DIS
LIN {X 0.251,Y -504.415,Z 274.536,A 0.000,B 0.000,C 90.000,E1 96.429} C_DIS
LIN {X -0.190,Y -505.886,Z 274.535,A 0.000,B 0.000,C 90.000,E1 96.258} C_DIS
LIN {X 0.245,Y -507.104,Z 274.533,A 0.000,B 0.000,C 90.000,E1 95.967} C_DIS
LIN {X 0.123,Y -507.989,Z 274.532,A 0.000,B 0.000,C 90.000,E1 95.739} C_DIS
LIN {X -0.053,Y -508.916,Z 274.529,A 0.000,B 0.000,C 90.000,E1 95.277} C_DIS
LIN {X -0.228,Y -508.829,Z 274.527,A 0.000,B 0.000,C 90.000,E1 94.816} C_DIS
LIN {X 0.068,Y -507.705,Z 274.524,A 0.000,B 0.000,C 90.000,E1 94.302} C_DIS
LIN {X -0.035,Y -506.697,Z 274.523,A 0.000,B 0.000,C 90.000,E1 94.073} C_DIS
LIN {X -0.102,Y -505.324,Z 274.521,A 0.000,B 0.000,C 90.000,E1 93.841} C_DIS
LIN {X 0.099,Y -499.778,Z 274.517,A 0.000,B 0.000,C 90.000,E1 93.094} C_DIS
LIN {X 0.099,Y -491.695,Z 274.512,A 0.000,B 0.000,C 90.000,E1 92.121} C_DIS
LIN {X -0.027,Y -470.446,Z 274.498,A 0.000,B 0.000,C 90.000,E1 89.656} C_DIS
LIN {X -0.034,Y -456.731,Z 274.488,A 0.000,B 0.000,C 90.000,E1 87.879} C_DIS
LIN {X 0.090,Y -440.719,Z 274.475,A 0.000,B 0.000,C 90.000,E1 85.527} C_DIS
LIN {X 0.153,Y -422.806,Z 274.459,A 0.000,B 0.000,C 90.000,E1 82.591} C_DIS
LIN {X -0.062,Y -405.422,Z 274.441,A 0.000,B 0.000,C 90.000,E1 79.342} C_DIS
LIN {X 0.112,Y -396.870,Z 274.431,A 0.000,B 0.000,C 90.000,E1 77.645} C_DIS
LIN {X -0.065,Y -385.447,Z 274.419,A 0.000,B 0.000,C 90.000,E1 75.408} C_DIS
LIN {X 0.048,Y -375.622,Z 274.408,A 0.000,B 0.000,C 90.000,E1 73.378} C_DIS
LIN {X 0.071,Y -365.711,Z 274.396,A 0.000,B 0.000,C 90.000,E1 71.329} C_DIS
LIN {X 0.026,Y -351.855,Z 274.380,A 0.000,B 0.000,C 90.000,E1 68.358} C_DIS
LIN {X -0.098,Y -336.408,Z 274.359,A 0.000,B 0.000,C 90.000,E1 64.717} C_DIS
LIN {X 0.116,Y -322.422,Z 274.339,A 0.000,B 0.000,C 90.000,E1 60.923} C_DIS
LIN {X -0.167,Y -314.635,Z 274.326,A 0.000,B 0.000,C 90.000,E1 58.742} C_DIS
LIN {X -0.007,Y -305.001,Z 274.310,A 0.000,B 0.000,C 90.000,E1 55.801} C_DIS
LIN {X 0.017,Y -298.772,Z 274.299,A 0.000,B 0.000,C 90.000,E1 53.829} C_DIS
LIN {X 0.023,Y -290.543,Z 274.284,A 0.000,B 0.000,C 90.000,E1 51.170} C_DIS
LIN {X 0.087,Y -284.321,Z 274.273,A 0.000,B 0.000,C 90.000,E1 49.138} C_DIS
LIN {X 0.036,Y -274.129,Z 274.254,A 0.000,B 0.000,C 90.000,E1 45.729} C_DIS
LIN {X 0.103,Y -266.545,Z 274.239,A 0.000,B 0.000,C 90.000,E1 42.933} C_DIS
LIN {X 0.079,Y -260.983,Z 274.227,A 0.000,B 0.000,C 90.000,E1 40.825} C_DIS
LIN {X 0.010,Y -255.321,Z 274.215,A 0.000,B 0.000,C 90.000,E1 38.705} C_DIS
LIN {X 0.043,Y -249.558,Z 274.203,A 0.000,B 0.000,C 90.000,E1 36.537} C_DIS
LIN {X 0.022,Y -243.691,Z 274.191,A 0.000,B 0.000,C 90.000,E1 34.358} C_DIS
LIN {X -0.013,Y -234.137,Z 274.170,A 0.000,B 0.000,C 90.000,E1 30.669} C_DIS
LIN {X 0.059,Y -227.037,Z 274.154,A 0.000,B 0.000,C 90.000,E1 27.641} C_DIS
LIN {X 0.043,Y -220.734,Z 274.137,A 0.000,B 0.000,C 90.000,E1 24.591} C_DIS
LIN {X -0.028,Y -213.892,Z 274.115,A 0.000,B 0.000,C 90.000,E1 20.737} C_DIS
LIN {X -0.007,Y -208.039,Z 274.093,A 0.000,B 0.000,C 90.000,E1 16.804} C_DIS
LIN {X -0.005,Y -203.187,Z 274.071,A 0.000,B 0.000,C 90.000,E1 12.827} C_DIS
LIN {X 0.023,Y -199.352,Z 274.049,A 0.000,B 0.000,C 90.000,E1 8.803} C_DIS
LIN {X -0.058,Y -195.657,Z 274.017,A 0.000,B 0.000,C 90.000,E1 3.151} C_DIS
LIN {X 0.044,Y -193.646,Z 273.970,A 0.000,B 0.000,C 90.000,E1 354.609} C_DIS
LIN {X -0.083,Y -195.764,Z 273.925,A 0.000,B 0.000,C 90.000,E1 346.464} C_DIS
LIN {X -0.090,Y -198.955,Z 273.898,A 0.000,B 0.000,C 90.000,E1 341.583} C_DIS
LIN {X -0.078,Y -202.817,Z 273.875,A 0.000,B 0.000,C 90.000,E1 337.539} C_DIS
LIN {X 0.002,Y -207.689,Z 273.853,A 0.000,B 0.000,C 90.000,E1 333.512} C_DIS
LIN {X 0.055,Y -213.691,Z 273.831,A 0.000,B 0.000,C 90.000,E1 329.537} C_DIS
LIN {X 0.001,Y -219.393,Z 273.813,A 0.000,B 0.000,C 90.000,E1 326.421} C_DIS
LIN {X -0.030,Y -225.884,Z 273.796,A 0.000,B 0.000,C 90.000,E1 323.336} C_DIS
LIN {X 0.015,Y -233.296,Z 273.779,A 0.000,B 0.000,C 90.000,E1 320.275} C_DIS
LIN {X 0.012,Y -242.508,Z 273.761,A 0.000,B 0.000,C 90.000,E1 316.905} C_DIS
LIN {X -0.084,Y -252.774,Z 273.742,A 0.000,B 0.000,C 90.000,E1 313.623} C_DIS
LIN {X -0.043,Y -264.064,Z 273.724,A 0.000,B 0.000,C 90.000,E1 310.378} C_DIS
LIN {X -0.158,Y -276.544,Z 273.707,A 0.000,B 0.000,C 90.000,E1 307.237} C_DIS
LIN {X -0.111,Y -287.308,Z 273.693,A 0.000,B 0.000,C 90.000,E1 304.818} C_DIS
LIN {X 0.102,Y -301.025,Z 273.678,A 0.000,B 0.000,C 90.000,E1 302.084} C_DIS
LIN {X 0.004,Y -318.058,Z 273.662,A 0.000,B 0.000,C 90.000,E1 299.155} C_DIS
LIN {X 0.053,Y -338.636,Z 273.644,A 0.000,B 0.000,C 90.000,E1 295.976} C_DIS
LIN {X 0.026,Y -351.289,Z 273.634,A 0.000,B 0.000,C 90.000,E1 294.131} C_DIS
LIN {X -0.055,Y -363.993,Z 273.624,A 0.000,B 0.000,C 90.000,E1 292.333} C_DIS
LIN {X 0.192,Y -381.212,Z 273.611,A 0.000,B 0.000,C 90.000,E1 289.939} C_DIS
LIN {X 0.047,Y -394.422,Z 273.601,A 0.000,B 0.000,C 90.000,E1 288.236} C_DIS
LIN {X 0.008,Y -407.618,Z 273.592,A 0.000,B 0.000,C 90.000,E1 286.551} C_DIS
LIN {X 0.227,Y -422.870,Z 273.581,A 0.000,B 0.000,C 90.000,E1 284.592} C_DIS
LIN {X 0.027,Y -431.254,Z 273.575,A 0.000,B 0.000,C 90.000,E1 283.536} C_DIS
LIN {X 0.153,Y -436.995,Z 273.571,A 0.000,B 0.000,C 90.000,E1 282.715} C_DIS
LIN {X 0.123,Y -444.046,Z 273.565,A 0.000,B 0.000,C 90.000,E1 281.658} C_DIS
LIN {X 0.173,Y -450.638,Z 273.559,A 0.000,B 0.000,C 90.000,E1 280.602} C_DIS
LIN {X 0.031,Y -458.349,Z 273.552,A 0.000,B 0.000,C 90.000,E1 279.321} C_DIS
LIN {X -0.078,Y -465.563,Z 273.545,A 0.000,B 0.000,C 90.000,E1 278.049} C_DIS
LIN {X -0.078,Y -472.306,Z 273.538,A 0.000,B 0.000,C 90.000,E1 276.777} C_DIS
LIN {X 0.155,Y -477.107,Z 273.532,A 0.000,B 0.000,C 90.000,E1 275.739} C_DIS
LIN {X 0.106,Y -480.137,Z 273.528,A 0.000,B 0.000,C 90.000,E1 274.992} C_DIS
LIN {X -0.223,Y -481.770,Z 273.525,A 0.000,B 0.000,C 90.000,E1 274.531} C_DIS
LIN {X -0.063,Y -483.006,Z 273.522,A 0.000,B 0.000,C 90.000,E1 274.012} C_DIS
LIN {X 0.074,Y -483.885,Z 273.519,A 0.000,B 0.000,C 90.000,E1 273.498} C_DIS
LIN {X 0.248,Y -484.418,Z 273.517,A 0.000,B 0.000,C 90.000,E1 272.980} C_DIS
LIN {X -0.082,Y -484.645,Z 273.514,A 0.000,B 0.000,C 90.000,E1 272.522} C_DIS
LIN {X -0.230,Y -484.563,Z 273.508,A 0.000,B 0.000,C 90.000,E1 271.547} C_DIS
LIN {X -0.068,Y -484.318,Z 273.506,A 0.000,B 0.000,C 90.000,E1 271.031} C_DIS
LIN {X 0.094,Y -483.869,Z 273.503,A 0.000,B 0.000,C 90.000,E1 270.516} C_DIS
LIN {X -0.228,Y -483.085,Z 273.500,A 0.000,B 0.000,C 90.000,E1 270.057} C_DIS
LIN {X -0.069,Y -481.854,Z 273.497,A 0.000,B 0.000,C 90.000,E1 269.542} C_DIS
LIN {X 0.084,Y -480.088,Z 273.495,A 0.000,B 0.000,C 90.000,E1 269.026} C_DIS
LIN {X 0.227,Y -477.749,Z 273.492,A 0.000,B 0.000,C 90.000,E1 268.511} C_DIS
LIN {X -0.108,Y -474.693,Z 273.489,A 0.000,B 0.000,C 90.000,E1 268.051} C_DIS
LIN {X 0.004,Y -470.783,Z 273.486,A 0.000,B 0.000,C 90.000,E1 267.535} C_DIS
LIN {X -0.186,Y -468.475,Z 273.485,A 0.000,B 0.000,C 90.000,E1 267.306} C_DIS
LIN {X 0.014,Y -463.132,Z 273.482,A 0.000,B 0.000,C 90.000,E1 266.788} C_DIS
LIN {X -0.087,Y -460.061,Z 273.481,A 0.000,B 0.000,C 90.000,E1 266.560} C_DIS
LIN {X 0.043,Y -457.003,Z 273.480,A 0.000,B 0.000,C 90.000,E1 266.331} C_DIS
LIN {X 0.170,Y -453.480,Z 273.478,A 0.000,B 0.000,C 90.000,E1 266.102} C_DIS
LIN {X 0.148,Y -450.075,Z 273.478,A 0.000,B 0.000,C 90.000,E1 265.931} C_DIS
LIN {X 0.158,Y -446.084,Z 273.477,A 0.000,B 0.000,C 90.000,E1 265.755} C_DIS
LIN {X 0.020,Y -442.411,Z 273.476,A 0.000,B 0.000,C 90.000,E1 265.641} C_DIS
LIN {X 0.090,Y -433.792,Z 273.475,A 0.000,B 0.000,C 90.000,E1 265.412} C_DIS
LIN {X -0.046,Y -424.456,Z 273.474,A 0.000,B 0.000,C 90.000,E1 265.298} C_DIS
LIN {X 0.143,Y -419.123,Z 273.474,A 0.000,B 0.000,C 90.000,E1 265.241} C_DIS
LIN {X 0.037,Y -180.901,Z 273.474,A 0.000,B 0.000,C 90.000,E1 265.241} C_DIS
LIN {X 0.079,Y -180.288,Z 273.465,A 0.000,B 0.000,C 90.000,E1 263.685} C_DIS
LIN {X 0.066,Y -178.940,Z 273.443,A 0.000,B 0.000,C 90.000,E1 259.803} C_DIS
LIN {X -0.066,Y -175.989,Z 273.415,A 0.000,B 0.000,C 90.000,E1 254.755} C_DIS
LIN {X 0.048,Y -175.489,Z 273.410,A 0.000,B 0.000,C 90.000,E1 253.866} C_DIS
LIN {X -0.057,Y -172.234,Z 273.387,A 0.000,B 0.000,C 90.000,E1 249.625} C_DIS
LIN {X -0.079,Y -171.711,Z 273.382,A 0.000,B 0.000,C 90.000,E1 248.773} C_DIS
LIN {X 0.006,Y -167.306,Z 273.353,A 0.000,B 0.000,C 90.000,E1 243.563} C_DIS
LIN {X 0.012,Y -166.686,Z 273.348,A 0.000,B 0.000,C 90.000,E1 242.692} C_DIS
LIN {X 0.003,Y -162.668,Z 273.324,A 0.000,B 0.000,C 90.000,E1 238.329} C_DIS
LIN {X -0.024,Y -161.357,Z 273.314,A 0.000,B 0.000,C 90.000,E1 236.580} C_DIS
LIN {X 0.010,Y -157.350,Z 273.290,A 0.000,B 0.000,C 90.000,E1 232.145} C_DIS
LIN {X 0.039,Y -155.339,Z 273.275,A 0.000,B 0.000,C 90.000,E1 229.461} C_DIS
LIN {X -0.031,Y -151.687,Z 273.250,A 0.000,B 0.000,C 90.000,E1 225.000} C_DIS
LIN {X 0.017,Y -150.550,Z 273.240,A 0.000,B 0.000,C 90.000,E1 223.176} C_DIS
LIN {X 0.050,Y -147.277,Z 273.215,A 0.000,B 0.000,C 90.000,E1 218.624} C_DIS
LIN {X 0.022,Y -145.304,Z 273.194,A 0.000,B 0.000,C 90.000,E1 214.978} C_DIS
LIN {X 0.014,Y -142.397,Z 273.164,A 0.000,B 0.000,C 90.000,E1 209.461} C_DIS
LIN {X -0.003,Y -141.378,Z 273.148,A 0.000,B 0.000,C 90.000,E1 206.693} C_DIS
LIN {X 0.038,Y -139.348,Z 273.112,A 0.000,B 0.000,C 90.000,E1 200.174} C_DIS
LIN {X -0.020,Y -138.784,Z 273.097,A 0.000,B 0.000,C 90.000,E1 197.402} C_DIS
LIN {X 0.038,Y -138.344,Z 273.055,A 0.000,B 0.000,C 90.000,E1 189.905} C_DIS
LIN {X 0.058,Y -139.389,Z 273.008,A 0.000,B 0.000,C 90.000,E1 181.489} C_DIS
LIN {X -0.028,Y -141.286,Z 272.972,A 0.000,B 0.000,C 90.000,E1 175.008} C_DIS
LIN {X -0.070,Y -142.650,Z 272.957,A 0.000,B 0.000,C 90.000,E1 172.243} C_DIS
LIN {X 0.021,Y -144.988,Z 272.931,A 0.000,B 0.000,C 90.000,E1 167.589} C_DIS
LIN {X 0.012,Y -147.614,Z 272.911,A 0.000,B 0.000,C 90.000,E1 163.921} C_DIS
LIN {X -0.052,Y -150.238,Z 272.890,A 0.000,B 0.000,C 90.000,E1 160.296} C_DIS
LIN {X -0.036,Y -153.632,Z 272.870,A 0.000,B 0.000,C 90.000,E1 156.666} C_DIS
LIN {X 0.022,Y -157.046,Z 272.850,A 0.000,B 0.000,C 90.000,E1 153.050} C_DIS
LIN {X 0.021,Y -161.173,Z 272.831,A 0.000,B 0.000,C 90.000,E1 149.488} C_DIS
LIN {X -0.036,Y -163.269,Z 272.821,A 0.000,B 0.000,C 90.000,E1 147.740} C_DIS
LIN {X 0.062,Y -167.709,Z 272.801,A 0.000,B 0.000,C 90.000,E1 144.196} C_DIS
LIN {X -0.025,Y -171.529,Z 272.787,A 0.000,B 0.000,C 90.000,E1 141.618} C_DIS
LIN {X 0.018,Y -176.468,Z 272.768,A 0.000,B 0.000,C 90.000,E1 138.162} C_DIS
LIN {X 0.017,Y -180.765,Z 272.753,A 0.000,B 0.000,C 90.000,E1 135.607} C_DIS
LIN {X 0.006,Y -186.171,Z 272.735,A 0.000,B 0.000,C 90.000,E1 132.243} C_DIS
LIN {X 0.070,Y -190.808,Z 272.721,A 0.000,B 0.000,C 90.000,E1 129.725} C_DIS
LIN {X -0.011,Y -196.566,Z 272.703,A 0.000,B 0.000,C 90.000,E1 126.457} C_DIS
LIN {X 0.074,Y -201.337,Z 272.689,A 0.000,B 0.000,C 90.000,E1 123.992} C_DIS
LIN {X -0.045,Y -203.436,Z 272.682,A 0.000,B 0.000,C 90.000,E1 122.832} C_DIS
LIN {X -0.103,Y -305.625,Z 272.682,A 0.000,B 0.000,C 90.000,E1 122.832} C_DIS
LIN {X 0.075,Y -308.179,Z 272.682,A 0.000,B 0.000,C 90.000,E1 122.752} C_DIS
LIN {X -0.060,Y -311.971,Z 272.681,A 0.000,B 0.000,C 90.000,E1 122.594} C_DIS
LIN {X -0.101,Y -314.250,Z 272.680,A 0.000,B 0.000,C 90.000,E1 122.418} C_DIS
LIN {X 0.018,Y -318.121,Z 272.677,A 0.000,B 0.000,C 90.000,E1 121.926} C_DIS
LIN {X 0.082,Y -319.961,Z 272.676,A 0.000,B 0.000,C 90.000,E1 121.592} C_DIS
LIN {X -0.214,Y -322.593,Z 272.672,A 0.000,B 0.000,C 90.000,E1 121.003} C_DIS
LIN {X 0.092,Y -333.979,Z 272.656,A 0.000,B 0.000,C 90.000,E1 118.103} C_DIS
LIN {X -0.033,Y -346.801,Z 272.641,A 0.000,B 0.000,C 90.000,E1 115.335} C_DIS
LIN {X 0.025,Y -359.503,Z 272.627,A 0.000,B 0.000,C 90.000,E1 112.898} C_DIS
LIN {X -0.074,Y -373.528,Z 272.614,A 0.000,B 0.000,C 90.000,E1 110.536} C_DIS
LIN {X 0.139,Y -388.979,Z 272.601,A 0.000,B 0.000,C 90.000,E1 108.181} C_DIS
LIN {X -0.125,Y -405.972,Z 272.589,A 0.000,B 0.000,C 90.000,E1 105.953} C_DIS
LIN {X 0.093,Y -424.634,Z 272.576,A 0.000,B 0.000,C 90.000,E1 103.716} C_DIS
LIN {X -0.213,Y -444.629,Z 272.565,A 0.000,B 0.000,C 90.000,E1 101.658} C_DIS
LIN {X -0.153,Y -465.210,Z 272.554,A 0.000,B 0.000,C 90.000,E1 99.726} C_DIS
LIN {X -0.223,Y -488.967,Z 272.543,A 0.000,B 0.000,C 90.000,E1 97.757} C_DIS
LIN {X 0.189,Y -499.697,Z 272.538,A 0.000,B 0.000,C 90.000,E1 96.891} C_DIS
LIN {X -0.053,Y -502.159,Z 272.537,A 0.000,B 0.000,C 90.000,E1 96.720} C_DIS
LIN {X 0.262,Y -504.036,Z 272.536,A 0.000,B 0.000,C 90.000,E1 96.486} C_DIS
LIN {X 0.134,Y -505.788,Z 272.535,A 0.000,B 0.000,C 90.000,E1 96.258} C_DIS
LIN {X 0.006,Y -507.103,Z 272.534,A 0.000,B 0.000,C 90.000,E1 96.030} C_DIS
LIN {X -0.177,Y -508.731,Z 272.531,A 0.000,B 0.000,C 90.000,E1 95.568} C_DIS
LIN {X 0.154,Y -509.265,Z 272.528,A 0.000,B 0.000,C 90.000,E1 95.049} C_DIS
LIN {X -0.016,Y -508.789,Z 272.525,A 0.000,B 0.000,C 90.000,E1 94.588} C_DIS
LIN {X -0.221,Y -507.221,Z 272.523,A 0.000,B 0.000,C 90.000,E1 94.131} C_DIS
LIN {X 0.217,Y -505.939,Z 272.521,A 0.000,B 0.000,C 90.000,E1 93.841} C_DIS
LIN {X -0.104,Y -500.456,Z 272.517,A 0.000,B 0.000,C 90.000,E1 93.154} C_DIS
LIN {X -0.066,Y -492.405,Z 272.512,A 0.000,B 0.000,C 90.000,E1 92.178} C_DIS
LIN {X 0.012,Y -473.188,Z 272.500,A 0.000,B 0.000,C 90.000,E1 89.943} C_DIS
LIN {X 0.058,Y -459.225,Z 272.490,A 0.000,B 0.000,C 90.000,E1 88.165} C_DIS
LIN {X 0.029,Y -444.713,Z 272.478,A 0.000,B 0.000,C 90.000,E1 86.102} C_DIS
LIN {X -0.037,Y -424.887,Z 272.461,A 0.000,B 0.000,C 90.000,E1 82.932} C_DIS
LIN {X -0.123,Y -411.513,Z 272.447,A 0.000,B 0.000,C 90.000,E1 80.500} C_DIS
LIN {X 0.193,Y -401.669,Z 272.436,A 0.000,B 0.000,C 90.000,E1 78.522} C_DIS
LIN {X 0.038,Y -390.223,Z 272.424,A 0.000,B 0.000,C 90.000,E1 76.297} C_DIS
LIN {X -0.082,Y -377.575,Z 272.410,A 0.000,B 0.000,C 90.000,E1 73.740} C_DIS
LIN {X -0.044,Y -366.273,Z 272.397,A 0.000,B 0.000,C 90.000,E1 71.402} C_DIS
LIN {X 0.051,Y -352.435,Z 272.380,A 0.000,B 0.000,C 90.000,E1 68.411} C_DIS
LIN {X -0.189,Y -336.991,Z 272.360,A 0.000,B 0.000,C 90.000,E1 64.793} C_DIS
LIN {X 0.041,Y -322.976,Z 272.339,A 0.000,B 0.000,C 90.000,E1 61.001} C_DIS
LIN {X -0.066,Y -315.205,Z 272.327,A 0.000,B 0.000,C 90.000,E1 58.791} C_DIS
LIN {X -0.023,Y -304.487,Z 272.309,A 0.000,B 0.000,C 90.000,E1 55.548} C_DIS
LIN {X -0.014,Y -298.252,Z 272.298,A 0.000,B 0.000,C 90.000,E1 53.577} C_DIS
LIN {X -0.074,Y -290.024,Z 272.283,A 0.000,B 0.000,C 90.000,E1 50.928} C_DIS
LIN {X -0.014,Y -283.789,Z 272.272,A 0.000,B 0.000,C 90.000,E1 48.895} C_DIS
LIN {X -0.075,Y -273.645,Z 272.253,A 0.000,B 0.000,C 90.000,E1 45.486} C_DIS
LIN {X -0.017,Y -266.092,Z 272.237,A 0.000,B 0.000,C 90.000,E1 42.690} C_DIS
LIN {X 0.148,Y -260.488,Z 272.225,A 0.000,B 0.000,C 90.000,E1 40.539} C_DIS
LIN {X -0.129,Y -254.829,Z 272.214,A 0.000,B 0.000,C 90.000,E1 38.463} C_DIS
LIN {X -0.106,Y -249.049,Z 272.202,A 0.000,B 0.000,C 90.000,E1 36.297} C_DIS
LIN {X 0.062,Y -243.175,Z 272.189,A 0.000,B 0.000,C 90.000,E1 34.072} C_DIS
LIN {X 0.003,Y -233.697,Z 272.169,A 0.000,B 0.000,C 90.000,E1 30.384} C_DIS
LIN {X -0.049,Y -226.663,Z 272.152,A 0.000,B 0.000,C 90.000,E1 27.385} C_DIS
LIN {X -0.070,Y -220.446,Z 272.135,A 0.000,B 0.000,C 90.000,E1 24.335} C_DIS
LIN {X 0.049,Y -213.670,Z 272.114,A 0.000,B 0.000,C 90.000,E1 20.429} C_DIS
LIN {X 0.059,Y -207.907,Z 272.092,A 0.000,B 0.000,C 90.000,E1 16.496} C_DIS
LIN {X 0.002,Y -203.120,Z 272.070,A 0.000,B 0.000,C 90.000,E1 12.535} C_DIS
LIN {X 0.026,Y -199.360,Z 272.047,A 0.000,B 0.000,C 90.000,E1 8.511} C_DIS
LIN {X -0.073,Y -195.752,Z 272.016,A 0.000,B 0.000,C 90.000,E1 2.865} C_DIS
LIN {X -0.045,Y -196.389,Z 271.920,A 0.000,B 0.000,C 90.000,E1 345.644} C_DIS
LIN {X 0.083,Y -199.820,Z 271.893,A 0.000,B 0.000,C 90.000,E1 340.732} C_DIS
LIN {X -0.063,Y -203.894,Z 271.871,A 0.000,B 0.000,C 90.000,E1 336.741} C_DIS
LIN {X -0.053,Y -208.987,Z 271.848,A 0.000,B 0.000,C 90.000,E1 332.743} C_DIS
LIN {X 0.104,Y -213.885,Z 271.831,A 0.000,B 0.000,C 90.000,E1 329.537} C_DIS
LIN {X 0.056,Y -219.596,Z 271.814,A 0.000,B 0.000,C 90.000,E1 326.421} C_DIS
LIN {X 0.033,Y -226.108,Z 271.796,A 0.000,B 0.000,C 90.000,E1 323.336} C_DIS
LIN {X 0.086,Y -233.495,Z 271.779,A 0.000,B 0.000,C 90.000,E1 320.275} C_DIS
LIN {X 0.091,Y -242.713,Z 271.761,A 0.000,B 0.000,C 90.000,E1 316.905} C_DIS
LIN {X 0.004,Y -252.965,Z 271.742,A 0.000,B 0.000,C 90.000,E1 313.623} C_DIS
LIN {X 0.055,Y -264.258,Z 271.724,A 0.000,B 0.000,C 90.000,E1 310.378} C_DIS
LIN {X -0.051,Y -276.721,Z 271.707,A 0.000,B 0.000,C 90.000,E1 307.237} C_DIS
LIN {X 0.005,Y -287.501,Z 271.693,A 0.000,B 0.000,C 90.000,E1 304.818} C_DIS
LIN {X -0.026,Y -301.205,Z 271.678,A 0.000,B 0.000,C 90.000,E1 302.133} C_DIS
LIN {X -0.066,Y -320.213,Z 271.660,A 0.000,B 0.000,C 90.000,E1 298.871} C_DIS
LIN {X -0.097,Y -338.790,Z 271.645,A 0.000,B 0.000,C 90.000,E1 296.027} C_DIS
LIN {X 0.045,Y -351.408,Z 271.634,A 0.000,B 0.000,C 90.000,E1 294.155} C_DIS
LIN {X 0.116,Y -364.091,Z 271.624,A 0.000,B 0.000,C 90.000,E1 292.333} C_DIS
LIN {X 0.015,Y -381.238,Z 271.611,A 0.000,B 0.000,C 90.000,E1 289.993} C_DIS
LIN {X 0.235,Y -394.416,Z 271.602,A 0.000,B 0.000,C 90.000,E1 288.236} C_DIS
LIN {X 0.085,Y -407.582,Z 271.592,A 0.000,B 0.000,C 90.000,E1 286.567} C_DIS
LIN {X -0.089,Y -422.767,Z 271.581,A 0.000,B 0.000,C 90.000,E1 284.662} C_DIS
LIN {X 0.058,Y -429.083,Z 271.577,A 0.000,B 0.000,C 90.000,E1 283.828} C_DIS
LIN {X -0.070,Y -436.839,Z 271.571,A 0.000,B 0.000,C 90.000,E1 282.771} C_DIS
LIN {X -0.106,Y -443.901,Z 271.565,A 0.000,B 0.000,C 90.000,E1 281.715} C_DIS
LIN {X -0.064,Y -450.466,Z 271.559,A 0.000,B 0.000,C 90.000,E1 280.658} C_DIS
LIN {X 0.239,Y -458.143,Z 271.552,A 0.000,B 0.000,C 90.000,E1 279.321} C_DIS
LIN {X -0.158,Y -463.963,Z 271.546,A 0.000,B 0.000,C 90.000,E1 278.341} C_DIS
LIN {X -0.184,Y -470.828,Z 271.539,A 0.000,B 0.000,C 90.000,E1 277.068} C_DIS
LIN {X 0.035,Y -475.787,Z 271.534,A 0.000,B 0.000,C 90.000,E1 276.030} C_DIS
LIN {X 0.168,Y -478.014,Z 271.531,A 0.000,B 0.000,C 90.000,E1 275.511} C_DIS
LIN {X -0.164,Y -479.995,Z 271.528,A 0.000,B 0.000,C 90.000,E1 275.049} C_DIS
LIN {X -0.014,Y -481.648,Z 271.525,A 0.000,B 0.000,C 90.000,E1 274.531} C_DIS
LIN {X 0.144,Y -482.922,Z 271.522,A 0.000,B 0.000,C 90.000,E1 274.012} C_DIS
LIN {X -0.201,Y -483.819,Z 271.520,A 0.000,B 0.000,C 90.000,E1 273.555} C_DIS
LIN {X -0.029,Y -484.396,Z 271.517,A 0.000,B 0.000,C 90.000,E1 273.037} C_DIS
LIN {X 0.124,Y -484.687,Z 271.514,A 0.000,B 0.000,C 90.000,E1 272.522} C_DIS
LIN {X -0.023,Y -484.668,Z 271.509,A 0.000,B 0.000,C 90.000,E1 271.547} C_DIS
LIN {X 0.139,Y -484.426,Z 271.506,A 0.000,B 0.000,C 90.000,E1 271.031} C_DIS
LIN {X -0.183,Y -484.008,Z 271.503,A 0.000,B 0.000,C 90.000,E1 270.573} C_DIS
LIN {X -0.020,Y -483.223,Z 271.500,A 0.000,B 0.000,C 90.000,E1 270.057} C_DIS
LIN {X 0.139,Y -482.035,Z 271.498,A 0.000,B 0.000,C 90.000,E1 269.542} C_DIS
LIN {X -0.188,Y -480.293,Z 271.495,A 0.000,B 0.000,C 90.000,E1 269.083} C_DIS
LIN {X -0.042,Y -477.989,Z 271.492,A 0.000,B 0.000,C 90.000,E1 268.568} C_DIS
LIN {X 0.100,Y -474.944,Z 271.489,A 0.000,B 0.000,C 90.000,E1 268.051} C_DIS
LIN {X 0.211,Y -471.056,Z 271.486,A 0.000,B 0.000,C 90.000,E1 267.535} C_DIS
LIN {X -0.168,Y -466.261,Z 271.484,A 0.000,B 0.000,C 90.000,E1 267.078} C_DIS
LIN {X 0.026,Y -460.422,Z 271.481,A 0.000,B 0.000,C 90.000,E1 266.560} C_DIS
LIN {X 0.194,Y -453.728,Z 271.478,A 0.000,B 0.000,C 90.000,E1 266.102} C_DIS
LIN {X 0.143,Y -450.430,Z 271.478,A 0.000,B 0.000,C 90.000,E1 265.931} C_DIS
LIN {X 0.126,Y -446.362,Z 271.477,A 0.000,B 0.000,C 90.000,E1 265.755} C_DIS
LIN {X -0.014,Y -442.751,Z 271.476,A 0.000,B 0.000,C 90.000,E1 265.641} C_DIS
LIN {X 0.027,Y -434.264,Z 271.475,A 0.000,B 0.000,C 90.000,E1 265.412} C_DIS
LIN {X -0.135,Y -425.160,Z 271.474,A 0.000,B 0.000,C 90.000,E1 265.298} C_DIS
LIN {X -0.021,Y -417.190,Z 271.474,A 0.000,B 0.000,C 90.000,E1 265.241} C_DIS
LIN {X -0.035,Y -180.899,Z 271.474,A 0.000,B 0.000,C 90.000,E1 265.241} C_DIS
LIN {X 0.028,Y -180.281,Z 271.465,A 0.000,B 0.000,C 90.000,E1 263.685} C_DIS
LIN {X 0.016,Y -178.934,Z 271.443,A 0.000,B 0.000,C 90.000,E1 259.803} C_DIS
LIN {X 0.054,Y -175.982,Z 271.415,A 0.000,B 0.000,C 90.000,E1 254.700} C_DIS
LIN {X -0.001,Y -175.476,Z 271.410,A 0.000,B 0.000,C 90.000,E1 253.866} C_DIS
LIN {X 0.055,Y -172.223,Z 271.387,A 0.000,B 0.000,C 90.000,E1 249.571} C_DIS
LIN {X 0.033,Y -171.700,Z 271.382,A 0.000,B 0.000,C 90.000,E1 248.720} C_DIS
LIN {X -0.042,Y -167.294,Z 271.353,A 0.000,B 0.000,C 90.000,E1 243.563} C_DIS
LIN {X 0.041,Y -166.672,Z 271.348,A 0.000,B 0.000,C 90.000,E1 242.666} C_DIS
LIN {X -0.044,Y -162.654,Z 271.324,A 0.000,B 0.000,C 90.000,E1 238.329} C_DIS
LIN {X 0.019,Y -161.343,Z 271.314,A 0.000,B 0.000,C 90.000,E1 236.548} C_DIS
LIN {X 0.061,Y -157.338,Z 271.290,A 0.000,B 0.000,C 90.000,E1 232.110} C_DIS
LIN {X -0.006,Y -155.322,Z 271.275,A 0.000,B 0.000,C 90.000,E1 229.461} C_DIS
LIN {X -0.076,Y -151.675,Z 271.250,A 0.000,B 0.000,C 90.000,E1 225.000} C_DIS
LIN {X -0.028,Y -150.540,Z 271.240,A 0.000,B 0.000,C 90.000,E1 223.176} C_DIS
LIN {X 0.005,Y -147.265,Z 271.215,A 0.000,B 0.000,C 90.000,E1 218.624} C_DIS
LIN {X -0.021,Y -145.293,Z 271.194,A 0.000,B 0.000,C 90.000,E1 214.978} C_DIS
LIN {X -0.029,Y -142.391,Z 271.164,A 0.000,B 0.000,C 90.000,E1 209.461} C_DIS
LIN {X 0.016,Y -141.369,Z 271.148,A 0.000,B 0.000,C 90.000,E1 206.668} C_DIS
LIN {X -0.005,Y -139.345,Z 271.112,A 0.000,B 0.000,C 90.000,E1 200.174} C_DIS
LIN {X 0.000,Y -139.017,Z 271.102,A 0.000,B 0.000,C 90.000,E1 198.308} C_DIS
LIN {X -0.004,Y -138.342,Z 271.055,A 0.000,B 0.000,C 90.000,E1 189.905} C_DIS
LIN {X 0.015,Y -139.393,Z 271.008,A 0.000,B 0.000,C 90.000,E1 181.489} C_DIS
LIN {X 0.070,Y -141.294,Z 270.972,A 0.000,B 0.000,C 90.000,E1 174.951} C_DIS
LIN {X 0.027,Y -142.656,Z 270.957,A 0.000,B 0.000,C 90.000,E1 172.186} C_DIS
LIN {X -0.023,Y -144.998,Z 270.931,A 0.000,B 0.000,C 90.000,E1 167.589} C_DIS
LIN {X -0.033,Y -147.625,Z 270.911,A 0.000,B 0.000,C 90.000,E1 163.921} C_DIS
LIN {X 0.045,Y -150.252,Z 270.890,A 0.000,B 0.000,C 90.000,E1 160.242} C_DIS
LIN {X 0.059,Y -153.649,Z 270.870,A 0.000,B 0.000,C 90.000,E1 156.613} C_DIS
LIN {X -0.024,Y -157.064,Z 270.850,A 0.000,B 0.000,C 90.000,E1 153.050} C_DIS
LIN {X 0.055,Y -161.195,Z 270.830,A 0.000,B 0.000,C 90.000,E1 149.459} C_DIS
LIN {X 0.004,Y -163.287,Z 270.821,A 0.000,B 0.000,C 90.000,E1 147.709} C_DIS
LIN {X 0.014,Y -167.733,Z 270.801,A 0.000,B 0.000,C 90.000,E1 144.196} C_DIS
LIN {X -0.074,Y -171.551,Z 270.787,A 0.000,B 0.000,C 90.000,E1 141.618} C_DIS
LIN {X -0.033,Y -176.494,Z 270.768,A 0.000,B 0.000,C 90.000,E1 138.162} C_DIS
LIN {X 0.092,Y -180.792,Z 270.753,A 0.000,B 0.000,C 90.000,E1 135.567} C_DIS
LIN {X -0.046,Y -186.200,Z 270.735,A 0.000,B 0.000,C 90.000,E1 132.243} C_DIS
LIN {X 0.018,Y -190.837,Z 270.721,A 0.000,B 0.000,C 90.000,E1 129.725} C_DIS
LIN {X -0.065,Y -196.596,Z 270.702,A 0.000,B 0.000,C 90.000,E1 126.457} C_DIS
LIN {X 0.020,Y -201.362,Z 270.689,A 0.000,B 0.000,C 90.000,E1 123.992} C_DIS
LIN {X 0.063,Y -203.524,Z 270.682,A 0.000,B 0.000,C 90.000,E1 122.752} C_DIS
LIN {X 0.059,Y -305.423,Z 270.682,A 0.000,B 0.000,C 90.000,E1 122.752} C_DIS
LIN {X -0.011,Y -306.835,Z 270.682,A 0.000,B 0.000,C 90.000,E1 122.752} C_DIS
LIN {X 0.118,Y -311.596,Z 270.681,A 0.000,B 0.000,C 90.000,E1 122.546} C_DIS
LIN {X -0.184,Y -314.030,Z 270.680,A 0.000,B 0.000,C 90.000,E1 122.418} C_DIS
LIN {X 0.077,Y -317.878,Z 270.677,A 0.000,B 0.000,C 90.000,E1 121.926} C_DIS
LIN {X 0.034,Y -319.755,Z 270.676,A 0.000,B 0.000,C 90.000,E1 121.623} C_DIS
LIN {X -0.114,Y -321.228,Z 270.674,A 0.000,B 0.000,C 90.000,E1 121.337} C_DIS
LIN {X -0.018,Y -333.822,Z 270.656,A 0.000,B 0.000,C 90.000,E1 118.153} C_DIS
LIN {X 0.153,Y -346.626,Z 270.641,A 0.000,B 0.000,C 90.000,E1 115.335} C_DIS
LIN {X -0.117,Y -359.312,Z 270.627,A 0.000,B 0.000,C 90.000,E1 112.950} C_DIS
LIN {X -0.014,Y -373.320,Z 270.614,A 0.000,B 0.000,C 90.000,E1 110.556} C_DIS
LIN {X -0.037,Y -388.753,Z 270.601,A 0.000,B 0.000,C 90.000,E1 108.236} C_DIS
LIN {X -0.040,Y -405.725,Z 270.589,A 0.000,B 0.000,C 90.000,E1 105.969} C_DIS
LIN {X -0.120,Y -424.365,Z 270.576,A 0.000,B 0.000,C 90.000,E1 103.772} C_DIS
LIN {X -0.022,Y -444.350,Z 270.565,A 0.000,B 0.000,C 90.000,E1 101.658} C_DIS
LIN {X 0.030,Y -464.925,Z 270.554,A 0.000,B 0.000,C 90.000,E1 99.726} C_DIS
LIN {X -0.051,Y -488.675,Z 270.543,A 0.000,B 0.000,C 90.000,E1 97.757} C_DIS
LIN {X 0.116,Y -501.967,Z 270.537,A 0.000,B 0.000,C 90.000,E1 96.720} C_DIS
LIN {X -0.071,Y -503.952,Z 270.536,A 0.000,B 0.000,C 90.000,E1 96.543} C_DIS
LIN {X -0.185,Y -505.777,Z 270.535,A 0.000,B 0.000,C 90.000,E1 96.315} C_DIS
LIN {X 0.207,Y -507.146,Z 270.534,A 0.000,B 0.000,C 90.000,E1 96.030} C_DIS
LIN {X 0.026,Y -508.871,Z 270.531,A 0.000,B 0.000,C 90.000,E1 95.568} C_DIS
LIN {X -0.151,Y -509.490,Z 270.528,A 0.000,B 0.000,C 90.000,E1 95.106} C_DIS
LIN {X 0.188,Y -509.104,Z 270.526,A 0.000,B 0.000,C 90.000,E1 94.588} C_DIS
LIN {X -0.018,Y -507.639,Z 270.523,A 0.000,B 0.000,C 90.000,E1 94.131} C_DIS
LIN {X -0.084,Y -506.423,Z 270.522,A 0.000,B 0.000,C 90.000,E1 93.898} C_DIS
LIN {X 0.209,Y -502.938,Z 270.519,A 0.000,B 0.000,C 90.000,E1 93.383} C_DIS
LIN {X -0.227,Y -495.081,Z 270.514,A 0.000,B 0.000,C 90.000,E1 92.465} C_DIS
LIN {X 0.087,Y -484.379,Z 270.507,A 0.000,B 0.000,C 90.000,E1 91.203} C_DIS
LIN {X -0.040,Y -465.580,Z 270.494,A 0.000,B 0.000,C 90.000,E1 88.969} C_DIS
LIN {X 0.072,Y -450.494,Z 270.483,A 0.000,B 0.000,C 90.000,E1 86.906} C_DIS
LIN {X 0.147,Y -430.096,Z 270.465,A 0.000,B 0.000,C 90.000,E1 83.742} C_DIS
LIN {X 0.126,Y -416.224,Z 270.452,A 0.000,B 0.000,C 90.000,E1 81.319} C_DIS
LIN {X -0.058,Y -403.490,Z 270.438,A 0.000,B 0.000,C 90.000,E1 78.870} C_DIS
LIN {X -0.158,Y -392.057,Z 270.426,A 0.000,B 0.000,C 90.000,E1 76.645} C_DIS
LIN {X 0.049,Y -379.414,Z 270.411,A 0.000,B 0.000,C 90.000,E1 74.047} C_DIS
LIN {X 0.138,Y -369.549,Z 270.400,A 0.000,B 0.000,C 90.000,E1 72.000} C_DIS
LIN {X 0.087,Y -358.359,Z 270.387,A 0.000,B 0.000,C 90.000,E1 69.645} C_DIS
LIN {X -0.122,Y -345.031,Z 270.370,A 0.000,B 0.000,C 90.000,E1 66.666} C_DIS
LIN {X -0.002,Y -331.479,Z 270.351,A 0.000,B 0.000,C 90.000,E1 63.256} C_DIS
LIN {X -0.032,Y -319.074,Z 270.332,A 0.000,B 0.000,C 90.000,E1 59.793} C_DIS
LIN {X -0.102,Y -309.194,Z 270.316,A 0.000,B 0.000,C 90.000,E1 56.914} C_DIS
LIN {X 0.054,Y -300.820,Z 270.302,A 0.000,B 0.000,C 90.000,E1 54.276} C_DIS
LIN {X 0.105,Y -292.527,Z 270.287,A 0.000,B 0.000,C 90.000,E1 51.618} C_DIS
LIN {X 0.017,Y -286.348,Z 270.276,A 0.000,B 0.000,C 90.000,E1 49.622} C_DIS
LIN {X 0.007,Y -278.055,Z 270.261,A 0.000,B 0.000,C 90.000,E1 46.905} C_DIS
LIN {X -0.056,Y -268.379,Z 270.241,A 0.000,B 0.000,C 90.000,E1 43.461} C_DIS
LIN {X -0.045,Y -262.803,Z 270.230,A 0.000,B 0.000,C 90.000,E1 41.353} C_DIS
LIN {X 0.083,Y -257.155,Z 270.218,A 0.000,B 0.000,C 90.000,E1 39.197} C_DIS
LIN {X -0.056,Y -251.408,Z 270.206,A 0.000,B 0.000,C 90.000,E1 37.076} C_DIS
LIN {X -0.047,Y -245.579,Z 270.194,A 0.000,B 0.000,C 90.000,E1 34.898} C_DIS
LIN {X -0.025,Y -235.983,Z 270.173,A 0.000,B 0.000,C 90.000,E1 31.209} C_DIS
LIN {X -0.103,Y -228.754,Z 270.157,A 0.000,B 0.000,C 90.000,E1 28.231} C_DIS
LIN {X 0.027,Y -222.321,Z 270.140,A 0.000,B 0.000,C 90.000,E1 25.155} C_DIS
LIN {X 0.084,Y -215.381,Z 270.118,A 0.000,B 0.000,C 90.000,E1 21.280} C_DIS
LIN {X -0.055,Y -209.380,Z 270.097,A 0.000,B 0.000,C 90.000,E1 17.402} C_DIS
LIN {X 0.039,Y -204.354,Z 270.075,A 0.000,B 0.000,C 90.000,E1 13.411} C_DIS
LIN {X -0.065,Y -200.355,Z 270.052,A 0.000,B 0.000,C 90.000,E1 9.434} C_DIS
LIN {X 0.090,Y -196.463,Z 270.021,A 0.000,B 0.000,C 90.000,E1 3.726} C_DIS
LIN {X -0.037,Y -194.140,Z 269.979,A 0.000,B 0.000,C 90.000,E1 356.274} C_DIS
LIN {X -0.055,Y -195.810,Z 269.929,A 0.000,B 0.000,C 90.000,E1 347.285} C_DIS
LIN {X 0.080,Y -198.706,Z 269.902,A 0.000,B 0.000,C 90.000,E1 342.362} C_DIS
LIN {X 0.020,Y -202.305,Z 269.880,A 0.000,B 0.000,C 90.000,E1 338.337} C_DIS
LIN {X 0.004,Y -206.977,Z 269.857,A 0.000,B 0.000,C 90.000,E1 334.332} C_DIS
LIN {X -0.062,Y -212.784,Z 269.835,A 0.000,B 0.000,C 90.000,E1 330.383} C_DIS
LIN {X -0.069,Y -218.285,Z 269.818,A 0.000,B 0.000,C 90.000,E1 327.248} C_DIS
LIN {X 0.053,Y -224.611,Z 269.801,A 0.000,B 0.000,C 90.000,E1 324.116} C_DIS
LIN {X -0.073,Y -231.783,Z 269.784,A 0.000,B 0.000,C 90.000,E1 321.090} C_DIS
LIN {X 0.051,Y -240.789,Z 269.765,A 0.000,B 0.000,C 90.000,E1 317.676} C_DIS
LIN {X 0.088,Y -250.794,Z 269.747,A 0.000,B 0.000,C 90.000,E1 314.352} C_DIS
LIN {X -0.113,Y -261.840,Z 269.728,A 0.000,B 0.000,C 90.000,E1 311.148} C_DIS
LIN {X 0.047,Y -274.004,Z 269.711,A 0.000,B 0.000,C 90.000,E1 307.935} C_DIS
LIN {X -0.006,Y -286.075,Z 269.695,A 0.000,B 0.000,C 90.000,E1 305.185} C_DIS
LIN {X 0.092,Y -299.592,Z 269.680,A 0.000,B 0.000,C 90.000,E1 302.467} C_DIS
LIN {X -0.051,Y -316.485,Z 269.664,A 0.000,B 0.000,C 90.000,E1 299.539} C_DIS
LIN {X -0.062,Y -336.809,Z 269.646,A 0.000,B 0.000,C 90.000,E1 296.360} C_DIS
LIN {X 0.178,Y -347.316,Z 269.638,A 0.000,B 0.000,C 90.000,E1 294.771} C_DIS
LIN {X -0.104,Y -362.082,Z 269.626,A 0.000,B 0.000,C 90.000,E1 292.695} C_DIS
LIN {X 0.085,Y -379.076,Z 269.613,A 0.000,B 0.000,C 90.000,E1 290.301} C_DIS
LIN {X -0.103,Y -392.233,Z 269.603,A 0.000,B 0.000,C 90.000,E1 288.598} C_DIS
LIN {X -0.111,Y -407.547,Z 269.592,A 0.000,B 0.000,C 90.000,E1 286.622} C_DIS
LIN {X 0.112,Y -422.663,Z 269.582,A 0.000,B 0.000,C 90.000,E1 284.662} C_DIS
LIN {X 0.014,Y -430.963,Z 269.576,A 0.000,B 0.000,C 90.000,E1 283.592} C_DIS
LIN {X 0.136,Y -436.686,Z 269.571,A 0.000,B 0.000,C 90.000,E1 282.771} C_DIS
LIN {X 0.101,Y -443.751,Z 269.565,A 0.000,B 0.000,C 90.000,E1 281.715} C_DIS
LIN {X 0.145,Y -450.267,Z 269.559,A 0.000,B 0.000,C 90.000,E1 280.658} C_DIS
LIN {X -0.004,Y -457.967,Z 269.552,A 0.000,B 0.000,C 90.000,E1 279.378} C_DIS
LIN {X -0.122,Y -465.169,Z 269.545,A 0.000,B 0.000,C 90.000,E1 278.106} C_DIS
LIN {X -0.129,Y -471.935,Z 269.538,A 0.000,B 0.000,C 90.000,E1 276.834} C_DIS
LIN {X 0.098,Y -476.756,Z 269.532,A 0.000,B 0.000,C 90.000,E1 275.796} C_DIS
LIN {X 0.046,Y -479.813,Z 269.528,A 0.000,B 0.000,C 90.000,E1 275.049} C_DIS
LIN {X 0.194,Y -481.508,Z 269.525,A 0.000,B 0.000,C 90.000,E1 274.531} C_DIS
LIN {X -0.163,Y -482.834,Z 269.523,A 0.000,B 0.000,C 90.000,E1 274.073} C_DIS
LIN {X 0.006,Y -483.796,Z 269.520,A 0.000,B 0.000,C 90.000,E1 273.555} C_DIS
LIN {X 0.179,Y -484.400,Z 269.517,A 0.000,B 0.000,C 90.000,E1 273.037} C_DIS
LIN {X -0.151,Y -484.721,Z 269.514,A 0.000,B 0.000,C 90.000,E1 272.579} C_DIS
LIN {X 0.008,Y -484.823,Z 269.511,A 0.000,B 0.000,C 90.000,E1 272.064} C_DIS
LIN {X -0.137,Y -484.544,Z 269.506,A 0.000,B 0.000,C 90.000,E1 271.088} C_DIS
LIN {X 0.027,Y -484.153,Z 269.503,A 0.000,B 0.000,C 90.000,E1 270.573} C_DIS
LIN {X 0.189,Y -483.400,Z 269.500,A 0.000,B 0.000,C 90.000,E1 270.057} C_DIS
LIN {X -0.133,Y -482.246,Z 269.498,A 0.000,B 0.000,C 90.000,E1 269.599} C_DIS
LIN {X 0.021,Y -480.567,Z 269.495,A 0.000,B 0.000,C 90.000,E1 269.083} C_DIS
LIN {X 0.167,Y -478.242,Z 269.492,A 0.000,B 0.000,C 90.000,E1 268.568} C_DIS
LIN {X -0.165,Y -475.218,Z 269.489,A 0.000,B 0.000,C 90.000,E1 268.108} C_DIS
LIN {X -0.050,Y -471.383,Z 269.487,A 0.000,B 0.000,C 90.000,E1 267.593} C_DIS
LIN {X 0.041,Y -466.600,Z 269.484,A 0.000,B 0.000,C 90.000,E1 267.078} C_DIS
LIN {X 0.235,Y -460.893,Z 269.481,A 0.000,B 0.000,C 90.000,E1 266.560} C_DIS
LIN {X -0.076,Y -454.381,Z 269.479,A 0.000,B 0.000,C 90.000,E1 266.159} C_DIS
LIN {X -0.163,Y -451.049,Z 269.478,A 0.000,B 0.000,C 90.000,E1 265.988} C_DIS
LIN {X 0.230,Y -447.067,Z 269.477,A 0.000,B 0.000,C 90.000,E1 265.755} C_DIS
LIN {X 0.045,Y -443.487,Z 269.476,A 0.000,B 0.000,C 90.000,E1 265.641} C_DIS
LIN {X -0.137,Y -439.040,Z 269.475,A 0.000,B 0.000,C 90.000,E1 265.527} C_DIS
LIN {X -0.001,Y -435.038,Z 269.475,A 0.000,B 0.000,C 90.000,E1 265.412} C_DIS
LIN {X -0.206,Y -425.832,Z 269.474,A 0.000,B 0.000,C 90.000,E1 265.298} C_DIS
LIN {X -0.098,Y -419.366,Z 269.473,A 0.000,B 0.000,C 90.000,E1 265.241} C_DIS
LIN {X -0.069,Y -180.897,Z 269.473,A 0.000,B 0.000,C 90.000,E1 265.241} C_DIS
LIN {X -0.006,Y -180.276,Z 269.465,A 0.000,B 0.000,C 90.000,E1 263.685} C_DIS
LIN {X -0.018,Y -178.930,Z 269.443,A 0.000,B 0.000,C 90.000,E1 259.803} C_DIS
LIN {X 0.019,Y -175.977,Z 269.415,A 0.000,B 0.000,C 90.000,E1 254.700} C_DIS
LIN {X -0.035,Y -175.467,Z 269.410,A 0.000,B 0.000,C 90.000,E1 253.866} C_DIS
LIN {X 0.022,Y -172.216,Z 269.387,A 0.000,B 0.000,C 90.000,E1 249.571} C_DIS
LIN {X -0.001,Y -171.693,Z 269.382,A 0.000,B 0.000,C 90.000,E1 248.720} C_DIS
LIN {X -0.010,Y -167.920,Z 269.358,A 0.000,B 0.000,C 90.000,E1 244.409} C_DIS
LIN {X 0.008,Y -166.662,Z 269.348,A 0.000,B 0.000,C 90.000,E1 242.666} C_DIS
LIN {X -0.076,Y -162.645,Z 269.324,A 0.000,B 0.000,C 90.000,E1 238.329} C_DIS
LIN {X -0.014,Y -161.333,Z 269.314,A 0.000,B 0.000,C 90.000,E1 236.548} C_DIS
LIN {X 0.029,Y -157.328,Z 269.290,A 0.000,B 0.000,C 90.000,E1 232.110} C_DIS
LIN {X -0.038,Y -155.311,Z 269.275,A 0.000,B 0.000,C 90.000,E1 229.461} C_DIS
LIN {X 0.000,Y -151.667,Z 269.250,A 0.000,B 0.000,C 90.000,E1 224.960} C_DIS
LIN {X 0.044,Y -150.533,Z 269.240,A 0.000,B 0.000,C 90.000,E1 223.137} C_DIS
LIN {X -0.025,Y -147.259,Z 269.215,A 0.000,B 0.000,C 90.000,E1 218.624} C_DIS
LIN {X 0.031,Y -145.284,Z 269.194,A 0.000,B 0.000,C 90.000,E1 214.945} C_DIS
LIN {X 0.065,Y -142.386,Z 269.164,A 0.000,B 0.000,C 90.000,E1 209.411} C_DIS
LIN {X -0.013,Y -141.364,Z 269.148,A 0.000,B 0.000,C 90.000,E1 206.668} C_DIS
LIN {X -0.035,Y -139.344,Z 269.112,A 0.000,B 0.000,C 90.000,E1 200.174} C_DIS
LIN {X -0.029,Y -139.013,Z 269.102,A 0.000,B 0.000,C 90.000,E1 198.308} C_DIS
LIN {X -0.033,Y -138.341,Z 269.055,A 0.000,B 0.000,C 90.000,E1 189.905} C_DIS
LIN {X -0.014,Y -139.397,Z 269.008,A 0.000,B 0.000,C 90.000,E1 181.489} C_DIS
LIN {X 0.040,Y -141.300,Z 268.972,A 0.000,B 0.000,C 90.000,E1 174.951} C_DIS
LIN {X -0.003,Y -142.661,Z 268.957,A 0.000,B 0.000,C 90.000,E1 172.186} C_DIS
LIN {X -0.053,Y -145.006,Z 268.931,A 0.000,B 0.000,C 90.000,E1 167.589} C_DIS
LIN {X -0.064,Y -147.632,Z 268.911,A 0.000,B 0.000,C 90.000,E1 163.921} C_DIS
LIN {X 0.014,Y -150.262,Z 268.890,A 0.000,B 0.000,C 90.000,E1 160.242} C_DIS
LIN {X 0.028,Y -153.662,Z 268.870,A 0.000,B 0.000,C 90.000,E1 156.613} C_DIS
LIN {X 0.084,Y -157.076,Z 268.850,A 0.000,B 0.000,C 90.000,E1 152.999} C_DIS
LIN {X 0.023,Y -161.210,Z 268.830,A 0.000,B 0.000,C 90.000,E1 149.459} C_DIS
LIN {X -0.029,Y -163.301,Z 268.821,A 0.000,B 0.000,C 90.000,E1 147.709} C_DIS
LIN {X -0.019,Y -167.748,Z 268.801,A 0.000,B 0.000,C 90.000,E1 144.196} C_DIS
LIN {X -0.001,Y -171.565,Z 268.787,A 0.000,B 0.000,C 90.000,E1 141.582} C_DIS
LIN {X -0.067,Y -176.511,Z 268.767,A 0.000,B 0.000,C 90.000,E1 138.162} C_DIS
LIN {X 0.058,Y -180.810,Z 268.753,A 0.000,B 0.000,C 90.000,E1 135.567} C_DIS
LIN {X 0.044,Y -186.218,Z 268.735,A 0.000,B 0.000,C 90.000,E1 132.204} C_DIS
LIN {X -0.018,Y -190.855,Z 268.721,A 0.000,B 0.000,C 90.000,E1 129.725} C_DIS
LIN {X 0.016,Y -196.617,Z 268.702,A 0.000,B 0.000,C 90.000,E1 126.423} C_DIS
LIN {X -0.071,Y -199.855,Z 268.693,A 0.000,B 0.000,C 90.000,E1 124.818} C_DIS
LIN {X 0.043,Y -203.623,Z 268.682,A 0.000,B 0.000,C 90.000,E1 122.704} C_DIS
LIN {X 0.033,Y -306.125,Z 268.682,A 0.000,B 0.000,C 90.000,E1 122.704} C_DIS
LIN {X 0.106,Y -307.392,Z 268.682,A 0.000,B 0.000,C 90.000,E1 122.673} C_DIS
LIN {X -0.066,Y -311.485,Z 268.681,A 0.000,B 0.000,C 90.000,E1 122.546} C_DIS
LIN {X 0.192,Y -313.730,Z 268.680,A 0.000,B 0.000,C 90.000,E1 122.339} C_DIS
LIN {X 0.136,Y -317.613,Z 268.677,A 0.000,B 0.000,C 90.000,E1 121.926} C_DIS
LIN {X -0.108,Y -319.517,Z 268.676,A 0.000,B 0.000,C 90.000,E1 121.671} C_DIS
LIN {X 0.088,Y -321.018,Z 268.674,A 0.000,B 0.000,C 90.000,E1 121.337} C_DIS
LIN {X -0.144,Y -334.996,Z 268.655,A 0.000,B 0.000,C 90.000,E1 117.897} C_DIS
LIN {X 0.053,Y -347.953,Z 268.639,A 0.000,B 0.000,C 90.000,E1 115.079} C_DIS
LIN {X 0.142,Y -360.780,Z 268.626,A 0.000,B 0.000,C 90.000,E1 112.642} C_DIS
LIN {X -0.058,Y -374.941,Z 268.613,A 0.000,B 0.000,C 90.000,E1 110.301} C_DIS
LIN {X -0.171,Y -390.539,Z 268.600,A 0.000,B 0.000,C 90.000,E1 108.000} C_DIS
LIN {X -0.019,Y -407.691,Z 268.587,A 0.000,B 0.000,C 90.000,E1 105.717} C_DIS
LIN {X -0.166,Y -426.524,Z 268.575,A 0.000,B 0.000,C 90.000,E1 103.536} C_DIS
LIN {X 0.070,Y -446.599,Z 268.564,A 0.000,B 0.000,C 90.000,E1 101.422} C_DIS
LIN {X 0.196,Y -467.233,Z 268.553,A 0.000,B 0.000,C 90.000,E1 99.500} C_DIS
LIN {X -0.173,Y -491.013,Z 268.542,A 0.000,B 0.000,C 90.000,E1 97.587} C_DIS
LIN {X -0.195,Y -501.716,Z 268.538,A 0.000,B 0.000,C 90.000,E1 96.777} C_DIS
LIN {X 0.058,Y -503.818,Z 268.536,A 0.000,B 0.000,C 90.000,E1 96.549} C_DIS
LIN {X 0.070,Y -505.685,Z 268.535,A 0.000,B 0.000,C 90.000,E1 96.315} C_DIS
LIN {X 0.026,Y -507.098,Z 268.534,A 0.000,B 0.000,C 90.000,E1 96.087} C_DIS
LIN {X -0.157,Y -508.976,Z 268.531,A 0.000,B 0.000,C 90.000,E1 95.625} C_DIS
LIN {X 0.173,Y -509.718,Z 268.528,A 0.000,B 0.000,C 90.000,E1 95.106} C_DIS
LIN {X 0.005,Y -509.448,Z 268.526,A 0.000,B 0.000,C 90.000,E1 94.645} C_DIS
LIN {X -0.199,Y -508.119,Z 268.523,A 0.000,B 0.000,C 90.000,E1 94.188} C_DIS
LIN {X 0.241,Y -506.986,Z 268.522,A 0.000,B 0.000,C 90.000,E1 93.898} C_DIS
LIN {X 0.140,Y -505.458,Z 268.520,A 0.000,B 0.000,C 90.000,E1 93.669} C_DIS
LIN {X 0.225,Y -497.821,Z 268.515,A 0.000,B 0.000,C 90.000,E1 92.694} C_DIS
LIN {X 0.221,Y -489.429,Z 268.510,A 0.000,B 0.000,C 90.000,E1 91.718} C_DIS
LIN {X -0.181,Y -466.218,Z 268.494,A 0.000,B 0.000,C 90.000,E1 89.026} C_DIS
LIN {X -0.050,Y -451.085,Z 268.483,A 0.000,B 0.000,C 90.000,E1 86.963} C_DIS
LIN {X -0.133,Y -432.262,Z 268.467,A 0.000,B 0.000,C 90.000,E1 84.090} C_DIS
LIN {X 0.050,Y -416.709,Z 268.452,A 0.000,B 0.000,C 90.000,E1 81.376} C_DIS
LIN {X -0.118,Y -403.949,Z 268.438,A 0.000,B 0.000,C 90.000,E1 78.926} C_DIS
LIN {X 0.181,Y -392.544,Z 268.426,A 0.000,B 0.000,C 90.000,E1 76.645} C_DIS
LIN {X 0.147,Y -378.530,Z 268.410,A 0.000,B 0.000,C 90.000,E1 73.795} C_DIS
LIN {X -0.143,Y -367.268,Z 268.397,A 0.000,B 0.000,C 90.000,E1 71.511} C_DIS
LIN {X -0.052,Y -354.833,Z 268.382,A 0.000,B 0.000,C 90.000,E1 68.827} C_DIS
LIN {X -0.025,Y -340.543,Z 268.364,A 0.000,B 0.000,C 90.000,E1 65.485} C_DIS
LIN {X -0.062,Y -327.421,Z 268.345,A 0.000,B 0.000,C 90.000,E1 62.076} C_DIS
LIN {X -0.023,Y -318.539,Z 268.331,A 0.000,B 0.000,C 90.000,E1 59.537} C_DIS
LIN {X 0.107,Y -307.605,Z 268.313,A 0.000,B 0.000,C 90.000,E1 56.294} C_DIS
LIN {X -0.026,Y -299.266,Z 268.298,A 0.000,B 0.000,C 90.000,E1 53.703} C_DIS
LIN {X -0.012,Y -290.983,Z 268.284,A 0.000,B 0.000,C 90.000,E1 51.045} C_DIS
LIN {X 0.055,Y -284.769,Z 268.272,A 0.000,B 0.000,C 90.000,E1 49.013} C_DIS
LIN {X 0.009,Y -274.584,Z 268.253,A 0.000,B 0.000,C 90.000,E1 45.607} C_DIS
LIN {X -0.102,Y -266.995,Z 268.238,A 0.000,B 0.000,C 90.000,E1 42.852} C_DIS
LIN {X 0.083,Y -261.392,Z 268.226,A 0.000,B 0.000,C 90.000,E1 40.701} C_DIS
LIN {X -0.014,Y -255.708,Z 268.214,A 0.000,B 0.000,C 90.000,E1 38.588} C_DIS
LIN {X 0.018,Y -249.944,Z 268.202,A 0.000,B 0.000,C 90.000,E1 36.423} C_DIS
LIN {X -0.005,Y -244.100,Z 268.190,A 0.000,B 0.000,C 90.000,E1 34.246} C_DIS
LIN {X 0.151,Y -236.471,Z 268.174,A 0.000,B 0.000,C 90.000,E1 31.258} C_DIS
LIN {X -0.036,Y -229.225,Z 268.157,A 0.000,B 0.000,C 90.000,E1 28.309} C_DIS
LIN {X -0.092,Y -222.795,Z 268.140,A 0.000,B 0.000,C 90.000,E1 25.283} C_DIS
LIN {X -0.015,Y -215.831,Z 268.119,A 0.000,B 0.000,C 90.000,E1 21.408} C_DIS
LIN {X -0.043,Y -210.907,Z 268.102,A 0.000,B 0.000,C 90.000,E1 18.290} C_DIS
LIN {X 0.093,Y -205.663,Z 268.080,A 0.000,B 0.000,C 90.000,E1 14.300} C_DIS
LIN {X 0.073,Y -201.420,Z 268.057,A 0.000,B 0.000,C 90.000,E1 10.310} C_DIS
LIN {X -0.070,Y -197.757,Z 268.031,A 0.000,B 0.000,C 90.000,E1 5.511} C_DIS
LIN {X -0.035,Y -194.982,Z 267.997,A 0.000,B 0.000,C 90.000,E1 359.542} C_DIS
LIN {X -0.015,Y -196.401,Z 267.925,A 0.000,B 0.000,C 90.000,E1 346.464} C_DIS
LIN {X 0.002,Y -199.516,Z 267.898,A 0.000,B 0.000,C 90.000,E1 341.583} C_DIS
LIN {X 0.033,Y -203.322,Z 267.875,A 0.000,B 0.000,C 90.000,E1 337.539} C_DIS
LIN {X -0.054,Y -208.243,Z 267.853,A 0.000,B 0.000,C 90.000,E1 333.563} C_DIS
LIN {X -0.012,Y -212.997,Z 267.835,A 0.000,B 0.000,C 90.000,E1 330.383} C_DIS
LIN {X -0.013,Y -218.484,Z 267.818,A 0.000,B 0.000,C 90.000,E1 327.248} C_DIS
LIN {X -0.015,Y -224.823,Z 267.801,A 0.000,B 0.000,C 90.000,E1 324.149} C_DIS
LIN {X -0.003,Y -231.999,Z 267.784,A 0.000,B 0.000,C 90.000,E1 321.090} C_DIS
LIN {X -0.031,Y -240.992,Z 267.765,A 0.000,B 0.000,C 90.000,E1 317.715} C_DIS
LIN {X -0.002,Y -250.995,Z 267.747,A 0.000,B 0.000,C 90.000,E1 314.393} C_DIS
LIN {X -0.015,Y -262.018,Z 267.729,A 0.000,B 0.000,C 90.000,E1 311.148} C_DIS
LIN {X -0.013,Y -274.191,Z 267.711,A 0.000,B 0.000,C 90.000,E1 307.971} C_DIS
LIN {X 0.155,Y -284.669,Z 267.698,A 0.000,B 0.000,C 90.000,E1 305.518} C_DIS
LIN {X 0.060,Y -298.004,Z 267.682,A 0.000,B 0.000,C 90.000,E1 302.832} C_DIS
LIN {X 0.030,Y -314.719,Z 267.666,A 0.000,B 0.000,C 90.000,E1 299.873} C_DIS
LIN {X -0.029,Y -334.868,Z 267.648,A 0.000,B 0.000,C 90.000,E1 296.693} C_DIS
LIN {X -0.122,Y -345.364,Z 267.640,A 0.000,B 0.000,C 90.000,E1 295.155} C_DIS
LIN {X -0.129,Y -360.049,Z 267.628,A 0.000,B 0.000,C 90.000,E1 293.025} C_DIS
LIN {X 0.153,Y -376.984,Z 267.615,A 0.000,B 0.000,C 90.000,E1 290.610} C_DIS
LIN {X 0.085,Y -392.223,Z 267.603,A 0.000,B 0.000,C 90.000,E1 288.598} C_DIS
LIN {X 0.007,Y -405.336,Z 267.594,A 0.000,B 0.000,C 90.000,E1 286.913} C_DIS
LIN {X 0.172,Y -420.383,Z 267.583,A 0.000,B 0.000,C 90.000,E1 284.954} C_DIS
LIN {X 0.048,Y -428.817,Z 267.577,A 0.000,B 0.000,C 90.000,E1 283.883} C_DIS
LIN {X -0.084,Y -436.566,Z 267.571,A 0.000,B 0.000,C 90.000,E1 282.827} C_DIS
LIN {X -0.127,Y -443.581,Z 267.565,A 0.000,B 0.000,C 90.000,E1 281.771} C_DIS
LIN {X -0.090,Y -450.112,Z 267.559,A 0.000,B 0.000,C 90.000,E1 280.715} C_DIS
LIN {X 0.205,Y -457.782,Z 267.552,A 0.000,B 0.000,C 90.000,E1 279.378} C_DIS
LIN {X 0.089,Y -464.982,Z 267.545,A 0.000,B 0.000,C 90.000,E1 278.106} C_DIS
LIN {X 0.080,Y -471.725,Z 267.538,A 0.000,B 0.000,C 90.000,E1 276.834} C_DIS
LIN {X -0.166,Y -476.568,Z 267.532,A 0.000,B 0.000,C 90.000,E1 275.853} C_DIS
LIN {X -0.223,Y -479.657,Z 267.528,A 0.000,B 0.000,C 90.000,E1 275.106} C_DIS
LIN {X -0.076,Y -481.379,Z 267.525,A 0.000,B 0.000,C 90.000,E1 274.588} C_DIS
LIN {X 0.047,Y -482.735,Z 267.523,A 0.000,B 0.000,C 90.000,E1 274.073} C_DIS
LIN {X 0.215,Y -483.746,Z 267.520,A 0.000,B 0.000,C 90.000,E1 273.555} C_DIS
LIN {X -0.096,Y -484.385,Z 267.517,A 0.000,B 0.000,C 90.000,E1 273.094} C_DIS
LIN {X 0.056,Y -484.734,Z 267.514,A 0.000,B 0.000,C 90.000,E1 272.579} C_DIS
LIN {X 0.216,Y -484.883,Z 267.512,A 0.000,B 0.000,C 90.000,E1 272.064} C_DIS
LIN {X 0.072,Y -484.661,Z 267.506,A 0.000,B 0.000,C 90.000,E1 271.088} C_DIS
LIN {X 0.235,Y -484.299,Z 267.503,A 0.000,B 0.000,C 90.000,E1 270.573} C_DIS
LIN {X -0.085,Y -483.584,Z 267.501,A 0.000,B 0.000,C 90.000,E1 270.115} C_DIS
LIN {X 0.076,Y -482.461,Z 267.498,A 0.000,B 0.000,C 90.000,E1 269.599} C_DIS
LIN {X 0.231,Y -480.807,Z 267.495,A 0.000,B 0.000,C 90.000,E1 269.083} C_DIS
LIN {X -0.101,Y -478.485,Z 267.492,A 0.000,B 0.000,C 90.000,E1 268.625} C_DIS
LIN {X 0.046,Y -475.505,Z 267.490,A 0.000,B 0.000,C 90.000,E1 268.108} C_DIS
LIN {X 0.160,Y -471.707,Z 267.487,A 0.000,B 0.000,C 90.000,E1 267.593} C_DIS
LIN {X -0.215,Y -467.004,Z 267.484,A 0.000,B 0.000,C 90.000,E1 267.135} C_DIS
LIN {X -0.090,Y -461.255,Z 267.481,A 0.000,B 0.000,C 90.000,E1 266.617} C_DIS
LIN {X 0.038,Y -454.854,Z 267.479,A 0.000,B 0.000,C 90.000,E1 266.159} C_DIS
LIN {X -0.076,Y -451.510,Z 267.478,A 0.000,B 0.000,C 90.000,E1 265.988} C_DIS
LIN {X -0.156,Y -447.648,Z 267.477,A 0.000,B 0.000,C 90.000,E1 265.812} C_DIS
LIN {X 0.057,Y -443.970,Z 267.476,A 0.000,B 0.000,C 90.000,E1 265.641} C_DIS
LIN {X -0.172,Y -439.488,Z 267.475,A 0.000,B 0.000,C 90.000,E1 265.527} C_DIS
LIN {X -0.062,Y -435.621,Z 267.474,A 0.000,B 0.000,C 90.000,E1 265.412} C_DIS
LIN {X 0.135,Y -426.407,Z 267.474,A 0.000,B 0.000,C 90.000,E1 265.241} C_DIS
LIN {X 0.184,Y -419.361,Z 267.473,A 0.000,B 0.000,C 90.000,E1 265.184} C_DIS
LIN {X 0.069,Y -180.896,Z 267.473,A 0.000,B 0.000,C 90.000,E1 265.179} C_DIS
LIN {X 0.003,Y -180.046,Z 267.462,A 0.000,B 0.000,C 90.000,E1 263.166} C_DIS
LIN {X -0.048,Y -178.926,Z 267.443,A 0.000,B 0.000,C 90.000,E1 259.803} C_DIS
LIN {X -0.010,Y -175.973,Z 267.415,A 0.000,B 0.000,C 90.000,E1 254.700} C_DIS
LIN {X -0.065,Y -175.459,Z 267.410,A 0.000,B 0.000,C 90.000,E1 253.866} C_DIS
LIN {X -0.007,Y -172.210,Z 267.387,A 0.000,B 0.000,C 90.000,E1 249.571} C_DIS
LIN {X -0.029,Y -171.686,Z 267.382,A 0.000,B 0.000,C 90.000,E1 248.720} C_DIS
LIN {X -0.039,Y -167.912,Z 267.358,A 0.000,B 0.000,C 90.000,E1 244.409} C_DIS
LIN {X -0.020,Y -166.654,Z 267.348,A 0.000,B 0.000,C 90.000,E1 242.666} C_DIS
LIN {X 0.034,Y -162.638,Z 267.324,A 0.000,B 0.000,C 90.000,E1 238.280} C_DIS
LIN {X -0.041,Y -161.325,Z 267.314,A 0.000,B 0.000,C 90.000,E1 236.548} C_DIS
LIN {X 0.002,Y -157.321,Z 267.289,A 0.000,B 0.000,C 90.000,E1 232.110} C_DIS
LIN {X -0.065,Y -155.301,Z 267.275,A 0.000,B 0.000,C 90.000,E1 229.461} C_DIS
LIN {X 0.082,Y -151.660,Z 267.250,A 0.000,B 0.000,C 90.000,E1 224.919} C_DIS
LIN {X 0.018,Y -150.527,Z 267.240,A 0.000,B 0.000,C 90.000,E1 223.137} C_DIS
LIN {X -0.051,Y -147.252,Z 267.214,A 0.000,B 0.000,C 90.000,E1 218.624} C_DIS
LIN {X 0.005,Y -145.277,Z 267.194,A 0.000,B 0.000,C 90.000,E1 214.945} C_DIS
LIN {X 0.039,Y -142.381,Z 267.163,A 0.000,B 0.000,C 90.000,E1 209.411} C_DIS
LIN {X -0.038,Y -141.359,Z 267.148,A 0.000,B 0.000,C 90.000,E1 206.668} C_DIS
LIN {X 0.071,Y -139.342,Z 267.112,A 0.000,B 0.000,C 90.000,E1 200.120} C_DIS
LIN {X -0.011,Y -139.010,Z 267.102,A 0.000,B 0.000,C 90.000,E1 198.290} C_DIS
LIN {X -0.059,Y -138.341,Z 267.055,A 0.000,B 0.000,C 90.000,E1 189.905} C_DIS
LIN {X -0.039,Y -139.400,Z 267.008,A 0.000,B 0.000,C 90.000,E1 181.489} C_DIS
LIN {X 0.014,Y -141.304,Z 266.972,A 0.000,B 0.000,C 90.000,E1 174.951} C_DIS
LIN {X -0.028,Y -142.665,Z 266.957,A 0.000,B 0.000,C 90.000,E1 172.186} C_DIS
LIN {X -0.079,Y -145.012,Z 266.931,A 0.000,B 0.000,C 90.000,E1 167.589} C_DIS
LIN {X 0.052,Y -147.639,Z 266.910,A 0.000,B 0.000,C 90.000,E1 163.866} C_DIS
LIN {X -0.012,Y -150.271,Z 266.890,A 0.000,B 0.000,C 90.000,E1 160.242} C_DIS
LIN {X 0.001,Y -153.672,Z 266.870,A 0.000,B 0.000,C 90.000,E1 156.613} C_DIS
LIN {X 0.057,Y -157.087,Z 266.850,A 0.000,B 0.000,C 90.000,E1 152.999} C_DIS
LIN {X -0.004,Y -161.222,Z 266.830,A 0.000,B 0.000,C 90.000,E1 149.459} C_DIS
LIN {X 0.081,Y -163.311,Z 266.820,A 0.000,B 0.000,C 90.000,E1 147.661} C_DIS
LIN {X -0.048,Y -167.761,Z 266.801,A 0.000,B 0.000,C 90.000,E1 144.196} C_DIS
LIN {X 0.104,Y -171.578,Z 266.786,A 0.000,B 0.000,C 90.000,E1 141.537} C_DIS
LIN {X -0.095,Y -176.526,Z 266.767,A 0.000,B 0.000,C 90.000,E1 138.162} C_DIS
LIN {X 0.028,Y -180.825,Z 266.753,A 0.000,B 0.000,C 90.000,E1 135.567} C_DIS
LIN {X 0.013,Y -186.235,Z 266.734,A 0.000,B 0.000,C 90.000,E1 132.204} C_DIS
LIN {X -0.048,Y -190.871,Z 266.721,A 0.000,B 0.000,C 90.000,E1 129.725} C_DIS
LIN {X -0.015,Y -196.634,Z 266.702,A 0.000,B 0.000,C 90.000,E1 126.423} C_DIS
LIN {X -0.102,Y -199.874,Z 266.693,A 0.000,B 0.000,C 90.000,E1 124.818} C_DIS
LIN {X -0.001,Y -203.702,Z 266.682,A 0.000,B 0.000,C 90.000,E1 122.673} C_DIS
LIN {X -0.056,Y -305.692,Z 266.681,A 0.000,B 0.000,C 90.000,E1 122.673} C_DIS
LIN {X 0.095,Y -307.550,Z 266.681,A 0.000,B 0.000,C 90.000,E1 122.625} C_DIS
LIN {X 0.143,Y -313.378,Z 266.680,A 0.000,B 0.000,C 90.000,E1 122.339} C_DIS
LIN {X -0.075,Y -316.439,Z 266.678,A 0.000,B 0.000,C 90.000,E1 122.084} C_DIS
LIN {X -0.096,Y -320.091,Z 266.675,A 0.000,B 0.000,C 90.000,E1 121.544} C_DIS
LIN {X -0.025,Y -321.603,Z 266.673,A 0.000,B 0.000,C 90.000,E1 121.209} C_DIS
LIN {X 0.081,Y -334.254,Z 266.656,A 0.000,B 0.000,C 90.000,E1 118.025} C_DIS
LIN {X -0.197,Y -347.120,Z 266.640,A 0.000,B 0.000,C 90.000,E1 115.283} C_DIS
LIN {X 0.010,Y -359.862,Z 266.627,A 0.000,B 0.000,C 90.000,E1 112.823} C_DIS
LIN {X 0.130,Y -373.932,Z 266.614,A 0.000,B 0.000,C 90.000,E1 110.429} C_DIS
LIN {X 0.002,Y -389.430,Z 266.601,A 0.000,B 0.000,C 90.000,E1 108.127} C_DIS
LIN {X 0.139,Y -406.475,Z 266.588,A 0.000,B 0.000,C 90.000,E1 105.843} C_DIS
LIN {X 0.078,Y -425.192,Z 266.576,A 0.000,B 0.000,C 90.000,E1 103.647} C_DIS
LIN {X 0.222,Y -445.227,Z 266.564,A 0.000,B 0.000,C 90.000,E1 101.535} C_DIS
LIN {X -0.201,Y -465.826,Z 266.554,A 0.000,B 0.000,C 90.000,E1 99.670} C_DIS
LIN {X -0.206,Y -489.571,Z 266.543,A 0.000,B 0.000,C 90.000,E1 97.701} C_DIS
LIN {X -0.030,Y -502.819,Z 266.537,A 0.000,B 0.000,C 90.000,E1 96.663} C_DIS
LIN {X -0.144,Y -506.339,Z 266.535,A 0.000,B 0.000,C 90.000,E1 96.258} C_DIS
LIN {X -0.218,Y -507.700,Z 266.533,A 0.000,B 0.000,C 90.000,E1 96.024} C_DIS
LIN {X 0.160,Y -508.701,Z 266.532,A 0.000,B 0.000,C 90.000,E1 95.739} C_DIS
LIN {X -0.013,Y -509.816,Z 266.529,A 0.000,B 0.000,C 90.000,E1 95.277} C_DIS
LIN {X -0.227,Y -509.898,Z 266.527,A 0.000,B 0.000,C 90.000,E1 94.821} C_DIS
LIN {X 0.119,Y -508.957,Z 266.524,A 0.000,B 0.000,C 90.000,E1 94.302} C_DIS
LIN {X -0.048,Y -506.818,Z 266.521,A 0.000,B 0.000,C 90.000,E1 93.841} C_DIS
LIN {X -0.249,Y -503.305,Z 266.519,A 0.000,B 0.000,C 90.000,E1 93.383} C_DIS
LIN {X -0.179,Y -495.406,Z 266.513,A 0.000,B 0.000,C 90.000,E1 92.407} C_DIS
LIN {X 0.134,Y -484.676,Z 266.506,A 0.000,B 0.000,C 90.000,E1 91.146} C_DIS
LIN {X -0.194,Y -463.835,Z 266.493,A 0.000,B 0.000,C 90.000,E1 88.682} C_DIS
LIN {X 0.114,Y -447.166,Z 266.480,A 0.000,B 0.000,C 90.000,E1 86.331} C_DIS
LIN {X 0.082,Y -427.128,Z 266.462,A 0.000,B 0.000,C 90.000,E1 83.166} C_DIS
LIN {X 0.042,Y -413.537,Z 266.449,A 0.000,B 0.000,C 90.000,E1 80.735} C_DIS
LIN {X -0.003,Y -403.675,Z 266.438,A 0.000,B 0.000,C 90.000,E1 78.814} C_DIS
LIN {X -0.043,Y -390.870,Z 266.424,A 0.000,B 0.000,C 90.000,E1 76.297} C_DIS
LIN {X -0.138,Y -378.290,Z 266.410,A 0.000,B 0.000,C 90.000,E1 73.740} C_DIS
LIN {X -0.082,Y -367.067,Z 266.397,A 0.000,B 0.000,C 90.000,E1 71.402} C_DIS
LIN {X -0.013,Y -354.680,Z 266.382,A 0.000,B 0.000,C 90.000,E1 68.720} C_DIS
LIN {X 0.139,Y -340.458,Z 266.363,A 0.000,B 0.000,C 90.000,E1 65.357} C_DIS
LIN {X -0.063,Y -327.393,Z 266.344,A 0.000,B 0.000,C 90.000,E1 61.975} C_DIS
LIN {X -0.066,Y -317.401,Z 266.328,A 0.000,B 0.000,C 90.000,E1 59.125} C_DIS
LIN {X 0.041,Y -306.533,Z 266.310,A 0.000,B 0.000,C 90.000,E1 55.881} C_DIS
LIN {X 0.089,Y -300.297,Z 266.300,A 0.000,B 0.000,C 90.000,E1 53.909} C_DIS
LIN {X 0.129,Y -291.996,Z 266.285,A 0.000,B 0.000,C 90.000,E1 51.251} C_DIS
LIN {X 0.029,Y -285.791,Z 266.274,A 0.000,B 0.000,C 90.000,E1 49.256} C_DIS
LIN {X 0.012,Y -275.587,Z 266.255,A 0.000,B 0.000,C 90.000,E1 45.850} C_DIS
LIN {X 0.058,Y -266.042,Z 266.235,A 0.000,B 0.000,C 90.000,E1 42.366} C_DIS
LIN {X 0.048,Y -260.441,Z 266.224,A 0.000,B 0.000,C 90.000,E1 40.253} C_DIS
LIN {X 0.132,Y -254.719,Z 266.212,A 0.000,B 0.000,C 90.000,E1 38.096} C_DIS
LIN {X -0.001,Y -248.950,Z 266.200,A 0.000,B 0.000,C 90.000,E1 35.964} C_DIS
LIN {X -0.035,Y -243.132,Z 266.188,A 0.000,B 0.000,C 90.000,E1 33.785} C_DIS
LIN {X 0.103,Y -235.559,Z 266.171,A 0.000,B 0.000,C 90.000,E1 30.797} C_DIS
LIN {X -0.104,Y -228.444,Z 266.155,A 0.000,B 0.000,C 90.000,E1 27.847} C_DIS
LIN {X 0.019,Y -222.155,Z 266.138,A 0.000,B 0.000,C 90.000,E1 24.771} C_DIS
LIN {X -0.012,Y -215.294,Z 266.116,A 0.000,B 0.000,C 90.000,E1 20.918} C_DIS
LIN {X 0.080,Y -210.463,Z 266.099,A 0.000,B 0.000,C 90.000,E1 17.764} C_DIS
LIN {X 0.010,Y -205.346,Z 266.077,A 0.000,B 0.000,C 90.000,E1 13.828} C_DIS
LIN {X -0.057,Y -201.239,Z 266.055,A 0.000,B 0.000,C 90.000,E1 9.849} C_DIS
LIN {X -0.006,Y -197.679,Z 266.028,A 0.000,B 0.000,C 90.000,E1 4.992} C_DIS
LIN {X -0.083,Y -195.019,Z 265.993,A 0.000,B 0.000,C 90.000,E1 358.740} C_DIS
LIN {X -0.011,Y -196.244,Z 265.929,A 0.000,B 0.000,C 90.000,E1 347.285} C_DIS
LIN {X 0.033,Y -199.712,Z 265.898,A 0.000,B 0.000,C 90.000,E1 341.583} C_DIS
LIN {X 0.072,Y -203.502,Z 265.875,A 0.000,B 0.000,C 90.000,E1 337.539} C_DIS
LIN {X -0.009,Y -208.424,Z 265.853,A 0.000,B 0.000,C 90.000,E1 333.563} C_DIS
LIN {X -0.035,Y -214.496,Z 265.831,A 0.000,B 0.000,C 90.000,E1 329.616} C_DIS
LIN {X -0.075,Y -220.200,Z 265.814,A 0.000,B 0.000,C 90.000,E1 326.501} C_DIS
LIN {X -0.089,Y -226.762,Z 265.797,A 0.000,B 0.000,C 90.000,E1 323.417} C_DIS
LIN {X -0.026,Y -234.122,Z 265.780,A 0.000,B 0.000,C 90.000,E1 320.356} C_DIS
LIN {X -0.007,Y -243.313,Z 265.761,A 0.000,B 0.000,C 90.000,E1 316.986} C_DIS
LIN {X -0.081,Y -253.533,Z 265.743,A 0.000,B 0.000,C 90.000,E1 313.704} C_DIS
LIN {X -0.017,Y -264.782,Z 265.725,A 0.000,B 0.000,C 90.000,E1 310.458} C_DIS
LIN {X 0.061,Y -277.267,Z 265.707,A 0.000,B 0.000,C 90.000,E1 307.282} C_DIS
LIN {X -0.040,Y -288.048,Z 265.694,A 0.000,B 0.000,C 90.000,E1 304.898} C_DIS
LIN {X -0.054,Y -301.712,Z 265.679,A 0.000,B 0.000,C 90.000,E1 302.212} C_DIS
LIN {X -0.143,Y -318.803,Z 265.663,A 0.000,B 0.000,C 90.000,E1 299.283} C_DIS
LIN {X -0.082,Y -339.225,Z 265.645,A 0.000,B 0.000,C 90.000,E1 296.104} C_DIS
LIN {X -0.102,Y -351.709,Z 265.635,A 0.000,B 0.000,C 90.000,E1 294.259} C_DIS
LIN {X 0.099,Y -362.241,Z 265.626,A 0.000,B 0.000,C 90.000,E1 292.717} C_DIS
LIN {X -0.040,Y -379.156,Z 265.613,A 0.000,B 0.000,C 90.000,E1 290.375} C_DIS
LIN {X -0.071,Y -394.384,Z 265.602,A 0.000,B 0.000,C 90.000,E1 288.362} C_DIS
LIN {X -0.112,Y -407.445,Z 265.593,A 0.000,B 0.000,C 90.000,E1 286.677} C_DIS
LIN {X 0.104,Y -422.417,Z 265.582,A 0.000,B 0.000,C 90.000,E1 284.717} C_DIS
LIN {X -0.166,Y -428.660,Z 265.577,A 0.000,B 0.000,C 90.000,E1 283.939} C_DIS
LIN {X -0.065,Y -434.532,Z 265.573,A 0.000,B 0.000,C 90.000,E1 283.119} C_DIS
LIN {X 0.089,Y -440.002,Z 265.568,A 0.000,B 0.000,C 90.000,E1 282.299} C_DIS
LIN {X 0.089,Y -446.733,Z 265.563,A 0.000,B 0.000,C 90.000,E1 281.243} C_DIS
LIN {X -0.109,Y -454.580,Z 265.555,A 0.000,B 0.000,C 90.000,E1 279.962} C_DIS
LIN {X 0.251,Y -461.977,Z 265.548,A 0.000,B 0.000,C 90.000,E1 278.624} C_DIS
LIN {X 0.200,Y -468.899,Z 265.541,A 0.000,B 0.000,C 90.000,E1 277.352} C_DIS
LIN {X -0.076,Y -474.038,Z 265.535,A 0.000,B 0.000,C 90.000,E1 276.372} C_DIS
LIN {X -0.156,Y -477.491,Z 265.531,A 0.000,B 0.000,C 90.000,E1 275.625} C_DIS
LIN {X -0.015,Y -479.481,Z 265.528,A 0.000,B 0.000,C 90.000,E1 275.106} C_DIS
LIN {X 0.131,Y -481.236,Z 265.526,A 0.000,B 0.000,C 90.000,E1 274.588} C_DIS
LIN {X -0.228,Y -482.607,Z 265.523,A 0.000,B 0.000,C 90.000,E1 274.131} C_DIS
LIN {X -0.061,Y -483.683,Z 265.520,A 0.000,B 0.000,C 90.000,E1 273.612} C_DIS
LIN {X 0.111,Y -484.353,Z 265.517,A 0.000,B 0.000,C 90.000,E1 273.094} C_DIS
LIN {X -0.221,Y -484.740,Z 265.514,A 0.000,B 0.000,C 90.000,E1 272.636} C_DIS
LIN {X -0.063,Y -484.922,Z 265.512,A 0.000,B 0.000,C 90.000,E1 272.121} C_DIS
LIN {X -0.207,Y -484.773,Z 265.506,A 0.000,B 0.000,C 90.000,E1 271.146} C_DIS
LIN {X -0.042,Y -484.434,Z 265.503,A 0.000,B 0.000,C 90.000,E1 270.630} C_DIS
LIN {X 0.121,Y -483.758,Z 265.501,A 0.000,B 0.000,C 90.000,E1 270.115} C_DIS
LIN {X -0.199,Y -482.663,Z 265.498,A 0.000,B 0.000,C 90.000,E1 269.656} C_DIS
LIN {X -0.042,Y -481.039,Z 265.495,A 0.000,B 0.000,C 90.000,E1 269.141} C_DIS
LIN {X 0.107,Y -478.769,Z 265.492,A 0.000,B 0.000,C 90.000,E1 268.625} C_DIS
LIN {X -0.223,Y -475.810,Z 265.490,A 0.000,B 0.000,C 90.000,E1 268.165} C_DIS
LIN {X -0.104,Y -472.060,Z 265.487,A 0.000,B 0.000,C 90.000,E1 267.650} C_DIS
LIN {X -0.008,Y -467.399,Z 265.484,A 0.000,B 0.000,C 90.000,E1 267.135} C_DIS
LIN {X -0.183,Y -464.739,Z 265.483,A 0.000,B 0.000,C 90.000,E1 266.906} C_DIS
LIN {X 0.193,Y -458.817,Z 265.480,A 0.000,B 0.000,C 90.000,E1 266.388} C_DIS
LIN {X 0.132,Y -452.238,Z 265.478,A 0.000,B 0.000,C 90.000,E1 265.988} C_DIS
LIN {X 0.045,Y -448.531,Z 265.477,A 0.000,B 0.000,C 90.000,E1 265.812} C_DIS
LIN {X 0.215,Y -444.954,Z 265.476,A 0.000,B 0.000,C 90.000,E1 265.641} C_DIS
LIN {X -0.060,Y -440.561,Z 265.475,A 0.000,B 0.000,C 90.000,E1 265.527} C_DIS
LIN {X 0.009,Y -436.684,Z 265.475,A 0.000,B 0.000,C 90.000,E1 265.412} C_DIS
LIN {X 0.060,Y -427.105,Z 265.474,A 0.000,B 0.000,C 90.000,E1 265.241} C_DIS
LIN {X 0.082,Y -419.286,Z 265.473,A 0.000,B 0.000,C 90.000,E1 265.179} C_DIS
LIN {X 0.010,Y -180.894,Z 265.473,A 0.000,B 0.000,C 90.000,E1 265.179} C_DIS
LIN {X -0.082,Y -179.500,Z 265.454,A 0.000,B 0.000,C 90.000,E1 261.781} C_DIS
LIN {X 0.079,Y -179.008,Z 265.445,A 0.000,B 0.000,C 90.000,E1 260.038} C_DIS
LIN {X -0.003,Y -178.619,Z 265.440,A 0.000,B 0.000,C 90.000,E1 259.218} C_DIS
LIN {X 0.065,Y -175.671,Z 265.412,A 0.000,B 0.000,C 90.000,E1 254.102} C_DIS
LIN {X -0.092,Y -172.388,Z 265.388,A 0.000,B 0.000,C 90.000,E1 249.880} C_DIS
LIN {X -0.075,Y -171.190,Z 265.379,A 0.000,B 0.000,C 90.000,E1 248.156} C_DIS
LIN {X -0.024,Y -167.481,Z 265.354,A 0.000,B 0.000,C 90.000,E1 243.819} C_DIS
LIN {X -0.016,Y -166.877,Z 265.350,A 0.000,B 0.000,C 90.000,E1 242.948} C_DIS
LIN {X -0.024,Y -162.183,Z 265.321,A 0.000,B 0.000,C 90.000,E1 237.709} C_DIS
LIN {X 0.033,Y -160.750,Z 265.311,A 0.000,B 0.000,C 90.000,E1 235.928} C_DIS
LIN {X 0.012,Y -157.549,Z 265.291,A 0.000,B 0.000,C 90.000,E1 232.396} C_DIS
LIN {X -0.050,Y -155.578,Z 265.276,A 0.000,B 0.000,C 90.000,E1 229.747} C_DIS
LIN {X 0.002,Y -151.862,Z 265.251,A 0.000,B 0.000,C 90.000,E1 225.243} C_DIS
LIN {X 0.016,Y -150.085,Z 265.236,A 0.000,B 0.000,C 90.000,E1 222.528} C_DIS
LIN {X -0.066,Y -146.888,Z 265.211,A 0.000,B 0.000,C 90.000,E1 218.016} C_DIS
LIN {X 0.039,Y -145.475,Z 265.196,A 0.000,B 0.000,C 90.000,E1 215.231} C_DIS
LIN {X -0.045,Y -142.886,Z 265.170,A 0.000,B 0.000,C 90.000,E1 210.669} C_DIS
LIN {X 0.012,Y -141.504,Z 265.150,A 0.000,B 0.000,C 90.000,E1 206.950} C_DIS
LIN {X 0.060,Y -139.390,Z 265.114,A 0.000,B 0.000,C 90.000,E1 200.429} C_DIS
LIN {X -0.019,Y -139.096,Z 265.103,A 0.000,B 0.000,C 90.000,E1 198.598} C_DIS
LIN {X -0.027,Y -138.354,Z 265.057,A 0.000,B 0.000,C 90.000,E1 190.197} C_DIS
LIN {X -0.035,Y -139.516,Z 265.005,A 0.000,B 0.000,C 90.000,E1 180.859} C_DIS
LIN {X 0.046,Y -141.170,Z 264.974,A 0.000,B 0.000,C 90.000,E1 175.241} C_DIS
LIN {X 0.018,Y -142.549,Z 264.958,A 0.000,B 0.000,C 90.000,E1 172.470} C_DIS
LIN {X -0.057,Y -144.824,Z 264.933,A 0.000,B 0.000,C 90.000,E1 167.881} C_DIS
LIN {X 0.072,Y -147.446,Z 264.912,A 0.000,B 0.000,C 90.000,E1 164.157} C_DIS
LIN {X -0.042,Y -150.027,Z 264.892,A 0.000,B 0.000,C 90.000,E1 160.550} C_DIS
LIN {X -0.036,Y -153.365,Z 264.872,A 0.000,B 0.000,C 90.000,E1 156.922} C_DIS
LIN {X 0.013,Y -155.898,Z 264.857,A 0.000,B 0.000,C 90.000,E1 154.204} C_DIS
LIN {X -0.089,Y -159.757,Z 264.837,A 0.000,B 0.000,C 90.000,E1 150.667} C_DIS
LIN {X -0.024,Y -161.997,Z 264.827,A 0.000,B 0.000,C 90.000,E1 148.869} C_DIS
LIN {X -0.004,Y -166.190,Z 264.807,A 0.000,B 0.000,C 90.000,E1 145.341} C_DIS
LIN {X 0.094,Y -171.205,Z 264.788,A 0.000,B 0.000,C 90.000,E1 141.823} C_DIS
LIN {X 0.018,Y -176.089,Z 264.769,A 0.000,B 0.000,C 90.000,E1 138.405} C_DIS
LIN {X -0.120,Y -180.349,Z 264.755,A 0.000,B 0.000,C 90.000,E1 135.891} C_DIS
LIN {X -0.012,Y -185.759,Z 264.736,A 0.000,B 0.000,C 90.000,E1 132.486} C_DIS
LIN {X -0.099,Y -190.371,Z 264.722,A 0.000,B 0.000,C 90.000,E1 130.011} C_DIS
LIN {X -0.054,Y -197.697,Z 264.699,A 0.000,B 0.000,C 90.000,E1 125.884} C_DIS
LIN {X -0.012,Y -200.946,Z 264.690,A 0.000,B 0.000,C 90.000,E1 124.246} C_DIS
LIN {X -0.036,Y -203.808,Z 264.681,A 0.000,B 0.000,C 90.000,E1 122.625} C_DIS
LIN {X -0.090,Y -306.505,Z 264.681,A 0.000,B 0.000,C 90.000,E1 122.625} C_DIS
LIN {X 0.083,Y -308.912,Z 264.681,A 0.000,B 0.000,C 90.000,E1 122.546} C_DIS
LIN {X 0.207,Y -312.672,Z 264.680,A 0.000,B 0.000,C 90.000,E1 122.339} C_DIS
LIN {X -0.104,Y -314.950,Z 264.679,A 0.000,B 0.000,C 90.000,E1 122.212} C_DIS
LIN {X 0.143,Y -318.115,Z 264.677,A 0.000,B 0.000,C 90.000,E1 121.799} C_DIS
LIN {X -0.012,Y -320.060,Z 264.675,A 0.000,B 0.000,C 90.000,E1 121.514} C_DIS
LIN {X -0.062,Y -321.582,Z 264.673,A 0.000,B 0.000,C 90.000,E1 121.209} C_DIS
LIN {X 0.051,Y -334.254,Z 264.656,A 0.000,B 0.000,C 90.000,E1 118.025} C_DIS
LIN {X -0.225,Y -347.120,Z 264.640,A 0.000,B 0.000,C 90.000,E1 115.283} C_DIS
LIN {X -0.019,Y -359.865,Z 264.627,A 0.000,B 0.000,C 90.000,E1 112.823} C_DIS
LIN {X 0.100,Y -373.935,Z 264.614,A 0.000,B 0.000,C 90.000,E1 110.429} C_DIS
LIN {X -0.028,Y -389.437,Z 264.601,A 0.000,B 0.000,C 90.000,E1 108.127} C_DIS
LIN {X 0.108,Y -406.483,Z 264.588,A 0.000,B 0.000,C 90.000,E1 105.843} C_DIS
LIN {X 0.045,Y -425.204,Z 264.576,A 0.000,B 0.000,C 90.000,E1 103.647} C_DIS
LIN {X 0.202,Y -445.224,Z 264.564,A 0.000,B 0.000,C 90.000,E1 101.535} C_DIS
LIN {X 0.237,Y -465.825,Z 264.554,A 0.000,B 0.000,C 90.000,E1 99.613} C_DIS
LIN {X 0.238,Y -489.599,Z 264.543,A 0.000,B 0.000,C 90.000,E1 97.644} C_DIS
LIN {X -0.051,Y -502.864,Z 264.537,A 0.000,B 0.000,C 90.000,E1 96.663} C_DIS
LIN {X 0.269,Y -504.803,Z 264.536,A 0.000,B 0.000,C 90.000,E1 96.429} C_DIS
LIN {X 0.143,Y -506.608,Z 264.535,A 0.000,B 0.000,C 90.000,E1 96.201} C_DIS
LIN {X 0.071,Y -507.962,Z 264.533,A 0.000,B 0.000,C 90.000,E1 95.967} C_DIS
LIN {X -0.160,Y -509.641,Z 264.531,A 0.000,B 0.000,C 90.000,E1 95.511} C_DIS
LIN {X 0.177,Y -510.218,Z 264.528,A 0.000,B 0.000,C 90.000,E1 94.992} C_DIS
LIN {X 0.011,Y -509.784,Z 264.525,A 0.000,B 0.000,C 90.000,E1 94.531} C_DIS
LIN {X -0.152,Y -508.267,Z 264.523,A 0.000,B 0.000,C 90.000,E1 94.069} C_DIS
LIN {X 0.252,Y -507.017,Z 264.521,A 0.000,B 0.000,C 90.000,E1 93.784} C_DIS
LIN {X 0.045,Y -503.507,Z 264.518,A 0.000,B 0.000,C 90.000,E1 93.326} C_DIS
LIN {X 0.113,Y -495.595,Z 264.513,A 0.000,B 0.000,C 90.000,E1 92.350} C_DIS
LIN {X -0.056,Y -484.872,Z 264.506,A 0.000,B 0.000,C 90.000,E1 91.146} C_DIS
LIN {X -0.177,Y -465.965,Z 264.494,A 0.000,B 0.000,C 90.000,E1 88.912} C_DIS
LIN {X -0.028,Y -450.867,Z 264.482,A 0.000,B 0.000,C 90.000,E1 86.846} C_DIS
LIN {X 0.038,Y -430.467,Z 264.465,A 0.000,B 0.000,C 90.000,E1 83.685} C_DIS
LIN {X 0.091,Y -416.565,Z 264.451,A 0.000,B 0.000,C 90.000,E1 81.254} C_DIS
LIN {X 0.146,Y -405.204,Z 264.439,A 0.000,B 0.000,C 90.000,E1 79.050} C_DIS
LIN {X 0.000,Y -395.205,Z 264.428,A 0.000,B 0.000,C 90.000,E1 77.117} C_DIS
LIN {X -0.114,Y -383.974,Z 264.416,A 0.000,B 0.000,C 90.000,E1 74.866} C_DIS
LIN {X -0.136,Y -375.622,Z 264.406,A 0.000,B 0.000,C 90.000,E1 73.142} C_DIS
LIN {X -0.027,Y -364.470,Z 264.393,A 0.000,B 0.000,C 90.000,E1 70.786} C_DIS
LIN {X 0.062,Y -349.612,Z 264.375,A 0.000,B 0.000,C 90.000,E1 67.486} C_DIS
LIN {X 0.008,Y -334.680,Z 264.355,A 0.000,B 0.000,C 90.000,E1 63.819} C_DIS
LIN {X -0.066,Y -322.081,Z 264.335,A 0.000,B 0.000,C 90.000,E1 60.383} C_DIS
LIN {X 0.087,Y -314.360,Z 264.323,A 0.000,B 0.000,C 90.000,E1 58.122} C_DIS
LIN {X 0.015,Y -303.668,Z 264.305,A 0.000,B 0.000,C 90.000,E1 54.895} C_DIS
LIN {X 0.011,Y -297.435,Z 264.294,A 0.000,B 0.000,C 90.000,E1 52.924} C_DIS
LIN {X 0.016,Y -291.220,Z 264.283,A 0.000,B 0.000,C 90.000,E1 50.928} C_DIS
LIN {X -0.090,Y -285.017,Z 264.272,A 0.000,B 0.000,C 90.000,E1 48.933} C_DIS
LIN {X 0.069,Y -274.881,Z 264.253,A 0.000,B 0.000,C 90.000,E1 45.486} C_DIS
LIN {X 0.153,Y -267.241,Z 264.237,A 0.000,B 0.000,C 90.000,E1 42.690} C_DIS
LIN {X -0.118,Y -259.740,Z 264.222,A 0.000,B 0.000,C 90.000,E1 39.930} C_DIS
LIN {X 0.063,Y -252.083,Z 264.206,A 0.000,B 0.000,C 90.000,E1 37.030} C_DIS
LIN {X -0.115,Y -246.302,Z 264.194,A 0.000,B 0.000,C 90.000,E1 34.898} C_DIS
LIN {X 0.034,Y -238.630,Z 264.177,A 0.000,B 0.000,C 90.000,E1 31.926} C_DIS
LIN {X 0.014,Y -231.302,Z 264.161,A 0.000,B 0.000,C 90.000,E1 28.949} C_DIS
LIN {X 0.005,Y -224.712,Z 264.144,A 0.000,B 0.000,C 90.000,E1 25.924} C_DIS
LIN {X 0.048,Y -218.900,Z 264.127,A 0.000,B 0.000,C 90.000,E1 22.845} C_DIS
LIN {X 0.037,Y -212.469,Z 264.105,A 0.000,B 0.000,C 90.000,E1 18.960} C_DIS
LIN {X 0.081,Y -207.081,Z 264.083,A 0.000,B 0.000,C 90.000,E1 15.009} C_DIS
LIN {X -0.092,Y -202.652,Z 264.061,A 0.000,B 0.000,C 90.000,E1 11.074} C_DIS
LIN {X 0.056,Y -199.280,Z 264.039,A 0.000,B 0.000,C 90.000,E1 7.011} C_DIS
LIN {X -0.074,Y -196.108,Z 264.008,A 0.000,B 0.000,C 90.000,E1 1.375} C_DIS
LIN {X 0.053,Y -197.232,Z 263.920,A 0.000,B 0.000,C 90.000,E1 345.644} C_DIS
LIN {X 0.026,Y -200.580,Z 263.893,A 0.000,B 0.000,C 90.000,E1 340.786} C_DIS
LIN {X -0.095,Y -204.601,Z 263.871,A 0.000,B 0.000,C 90.000,E1 336.794} C_DIS
LIN {X -0.057,Y -209.737,Z 263.849,A 0.000,B 0.000,C 90.000,E1 332.794} C_DIS
LIN {X -0.124,Y -216.034,Z 263.827,A 0.000,B 0.000,C 90.000,E1 328.869} C_DIS
LIN {X -0.001,Y -221.964,Z 263.810,A 0.000,B 0.000,C 90.000,E1 325.722} C_DIS
LIN {X 0.033,Y -228.755,Z 263.792,A 0.000,B 0.000,C 90.000,E1 322.637} C_DIS
LIN {X 0.084,Y -237.286,Z 263.774,A 0.000,B 0.000,C 90.000,E1 319.218} C_DIS
LIN {X 0.024,Y -246.799,Z 263.755,A 0.000,B 0.000,C 90.000,E1 315.891} C_DIS
LIN {X 0.059,Y -257.319,Z 263.737,A 0.000,B 0.000,C 90.000,E1 312.609} C_DIS
LIN {X 0.061,Y -268.963,Z 263.719,A 0.000,B 0.000,C 90.000,E1 309.402} C_DIS
LIN {X -0.073,Y -281.923,Z 263.702,A 0.000,B 0.000,C 90.000,E1 306.297} C_DIS
LIN {X -0.075,Y -293.213,Z 263.688,A 0.000,B 0.000,C 90.000,E1 303.913} C_DIS
LIN {X 0.087,Y -303.723,Z 263.677,A 0.000,B 0.000,C 90.000,E1 301.878} C_DIS
LIN {X 0.072,Y -320.938,Z 263.661,A 0.000,B 0.000,C 90.000,E1 298.949} C_DIS
LIN {X 0.075,Y -339.357,Z 263.645,A 0.000,B 0.000,C 90.000,E1 296.104} C_DIS
LIN {X 0.064,Y -351.812,Z 263.635,A 0.000,B 0.000,C 90.000,E1 294.259} C_DIS
LIN {X -0.007,Y -364.370,Z 263.625,A 0.000,B 0.000,C 90.000,E1 292.461} C_DIS
LIN {X -0.214,Y -379.191,Z 263.613,A 0.000,B 0.000,C 90.000,E1 290.429} C_DIS
LIN {X -0.091,Y -396.535,Z 263.601,A 0.000,B 0.000,C 90.000,E1 288.109} C_DIS
LIN {X -0.218,Y -409.533,Z 263.591,A 0.000,B 0.000,C 90.000,E1 286.441} C_DIS
LIN {X -0.104,Y -422.338,Z 263.582,A 0.000,B 0.000,C 90.000,E1 284.773} C_DIS
LIN {X 0.205,Y -430.531,Z 263.576,A 0.000,B 0.000,C 90.000,E1 283.647} C_DIS
LIN {X 0.094,Y -438.069,Z 263.570,A 0.000,B 0.000,C 90.000,E1 282.591} C_DIS
LIN {X 0.071,Y -444.914,Z 263.564,A 0.000,B 0.000,C 90.000,E1 281.535} C_DIS
LIN {X -0.157,Y -452.851,Z 263.557,A 0.000,B 0.000,C 90.000,E1 280.254} C_DIS
LIN {X 0.182,Y -460.366,Z 263.550,A 0.000,B 0.000,C 90.000,E1 278.916} C_DIS
LIN {X 0.106,Y -467.363,Z 263.543,A 0.000,B 0.000,C 90.000,E1 277.644} C_DIS
LIN {X -0.187,Y -472.584,Z 263.537,A 0.000,B 0.000,C 90.000,E1 276.663} C_DIS
LIN {X 0.052,Y -477.315,Z 263.531,A 0.000,B 0.000,C 90.000,E1 275.625} C_DIS
LIN {X 0.193,Y -479.311,Z 263.529,A 0.000,B 0.000,C 90.000,E1 275.106} C_DIS
LIN {X -0.141,Y -481.091,Z 263.526,A 0.000,B 0.000,C 90.000,E1 274.645} C_DIS
LIN {X -0.021,Y -482.503,Z 263.523,A 0.000,B 0.000,C 90.000,E1 274.131} C_DIS
LIN {X 0.146,Y -483.601,Z 263.520,A 0.000,B 0.000,C 90.000,E1 273.612} C_DIS
LIN {X -0.167,Y -484.311,Z 263.517,A 0.000,B 0.000,C 90.000,E1 273.151} C_DIS
LIN {X -0.016,Y -484.756,Z 263.515,A 0.000,B 0.000,C 90.000,E1 272.636} C_DIS
LIN {X 0.143,Y -484.954,Z 263.512,A 0.000,B 0.000,C 90.000,E1 272.121} C_DIS
LIN {X -0.001,Y -484.850,Z 263.506,A 0.000,B 0.000,C 90.000,E1 271.146} C_DIS
LIN {X 0.164,Y -484.559,Z 263.504,A 0.000,B 0.000,C 90.000,E1 270.630} C_DIS
LIN {X -0.156,Y -483.901,Z 263.501,A 0.000,B 0.000,C 90.000,E1 270.172} C_DIS
LIN {X 0.007,Y -482.878,Z 263.498,A 0.000,B 0.000,C 90.000,E1 269.656} C_DIS
LIN {X 0.165,Y -481.270,Z 263.495,A 0.000,B 0.000,C 90.000,E1 269.141} C_DIS
LIN {X -0.001,Y -480.265,Z 263.494,A 0.000,B 0.000,C 90.000,E1 268.912} C_DIS
LIN {X 0.142,Y -477.674,Z 263.491,A 0.000,B 0.000,C 90.000,E1 268.396} C_DIS
LIN {X -0.192,Y -474.367,Z 263.488,A 0.000,B 0.000,C 90.000,E1 267.936} C_DIS
LIN {X -0.083,Y -470.240,Z 263.486,A 0.000,B 0.000,C 90.000,E1 267.421} C_DIS
LIN {X 0.001,Y -465.155,Z 263.483,A 0.000,B 0.000,C 90.000,E1 266.906} C_DIS
LIN {X -0.127,Y -459.240,Z 263.480,A 0.000,B 0.000,C 90.000,E1 266.445} C_DIS
LIN {X -0.086,Y -455.967,Z 263.479,A 0.000,B 0.000,C 90.000,E1 266.216} C_DIS
LIN {X 0.074,Y -448.900,Z 263.477,A 0.000,B 0.000,C 90.000,E1 265.812} C_DIS
LIN {X 0.213,Y -445.381,Z 263.476,A 0.000,B 0.000,C 90.000,E1 265.641} C_DIS
LIN {X -0.090,Y -440.937,Z 263.475,A 0.000,B 0.000,C 90.000,E1 265.527} C_DIS
LIN {X -0.032,Y -437.016,Z 263.474,A 0.000,B 0.000,C 90.000,E1 265.412} C_DIS
LIN {X -0.032,Y -427.490,Z 263.474,A 0.000,B 0.000,C 90.000,E1 265.241} C_DIS
LIN {X -0.053,Y -418.309,Z 263.473,A 0.000,B 0.000,C 90.000,E1 265.179} C_DIS
LIN {X -0.046,Y -180.892,Z 263.473,A 0.000,B 0.000,C 90.000,E1 265.179} C_DIS
LIN {X 0.034,Y -179.005,Z 263.445,A 0.000,B 0.000,C 90.000,E1 260.038} C_DIS
LIN {X -0.047,Y -178.609,Z 263.440,A 0.000,B 0.000,C 90.000,E1 259.218} C_DIS
LIN {X 0.021,Y -175.661,Z 263.412,A 0.000,B 0.000,C 90.000,E1 254.102} C_DIS
LIN {X 0.026,Y -172.378,Z 263.388,A 0.000,B 0.000,C 90.000,E1 249.826} C_DIS
LIN {X 0.040,Y -171.175,Z 263.378,A 0.000,B 0.000,C 90.000,E1 248.103} C_DIS
LIN {X 0.084,Y -167.470,Z 263.354,A 0.000,B 0.000,C 90.000,E1 243.768} C_DIS
LIN {X 0.017,Y -166.866,Z 263.350,A 0.000,B 0.000,C 90.000,E1 242.922} C_DIS
LIN {X 0.071,Y -162.172,Z 263.320,A 0.000,B 0.000,C 90.000,E1 237.661} C_DIS
LIN {X -0.008,Y -160.735,Z 263.311,A 0.000,B 0.000,C 90.000,E1 235.928} C_DIS
LIN {X -0.029,Y -157.537,Z 263.291,A 0.000,B 0.000,C 90.000,E1 232.396} C_DIS
LIN {X 0.028,Y -155.564,Z 263.276,A 0.000,B 0.000,C 90.000,E1 229.703} C_DIS
LIN {X -0.038,Y -151.852,Z 263.251,A 0.000,B 0.000,C 90.000,E1 225.243} C_DIS
LIN {X -0.024,Y -150.073,Z 263.236,A 0.000,B 0.000,C 90.000,E1 222.528} C_DIS
LIN {X 0.010,Y -146.879,Z 263.211,A 0.000,B 0.000,C 90.000,E1 217.971} C_DIS
LIN {X -0.001,Y -145.465,Z 263.196,A 0.000,B 0.000,C 90.000,E1 215.231} C_DIS
